BEGIN
	REGION read me
	  // ============================================================================
	  // PROGRAM START COMMENT
	  // ============================================================================
	  // EN:
	  // FC_AutoProcessPopup handles popup visualization and editing of AutoProcess
	  // data based on index from HMI.
	  // The function provides:
	  //  - automatic data loading from AutoProcessData according to selected index,
	  //  - two-step confirmation for safe data overwrite (compare first, write second),
	  //  - automatic reset of edit mode when index is changed,
	  //  - delete functionality for selected record,
	  //  - status bits for HMI to visualize pending changes and confirmation dialogs,
	  //  - index range control (1..16).
	  //
	  // Data flow:
	  // AutoProcessData  -> ActualSHowingData  (display mode)
	  // ActualSHowingData -> AutoProcessData  (after double confirmation)
	  //
	  // Usage:
	  // Call cyclically 
	  // RMS index is taken from AutoProcess_HMI.IndexProcess.
	  //
	  // ----------------------------------------------------------------------------
	  // CZ:
	  // FC_AutoProcessPopup obsluhuje zobrazení a editaci dat AutoProcess podle
	  // indexu z HMI.
	  // Funkce zajišťuje:
	  //  - automatické načítání dat z AutoProcessData podle zvoleného indexu,
	  //  - dvoukrokové potvrzení zápisu (nejprve porovnání, poté zápis),
	  //  - automatické zrušení editace při změně indexu,
	  //  - mazání záznamu podle indexu,
	  //  - stavové bity pro HMI (čekající změna, potvrzovací dialog),
	  //  - kontrolu rozsahu indexu (1..16).
	  //
	  // Tok dat:
	  // AutoProcessData  -> ActualSHowingData  (zobrazení)
	  // ActualSHowingData -> AutoProcessData  (po potvrzení)
	  //
	  // Použití:
	  // Volat cyklicky 
	  // Index je čten z AutoProcess_HMI.IndexProcess.
	  // ============================================================================
	  
	  // Statement section REGION
	  
	END_REGION
	
	
	REGION IndexRangeCheck
	  // EN: Clamp index to range 1..16
	  // CZ: Oříznutí indexu do rozsahu 1..16
	  IF #idx < 1 THEN
	    #idx := 1;
	    "AutoProcess_HMI".IndexProcess := #idx;
	  ELSIF #idx > 16 THEN
	    #idx := 16;
	    "AutoProcess_HMI".IndexProcess := #idx;
	    
	  END_IF;
	END_REGION
	
	
	REGION IndexHandling
	  // ---------------------------------------------------------------------------
	  // EN: Detect index change and reset edit session
	  // CZ: Detekce změny indexu a zrušení editace
	  // ---------------------------------------------------------------------------
	  #idx := "AutoProcess_HMI".IndexProcess;
	  
	  IF #idx <> "AutoProcess_HMI".Data_handling.LastIndex THEN
	    "AutoProcess_HMI".Data_handling.UpdateData_switch := FALSE;
	    "AutoProcess_HMI".Data_handling.UpdateData_Confirm := FALSE;
	    "AutoProcess_HMI".Data_handling.FinalConfirm_Write := FALSE;
	    "AutoProcess_HMI".Data_handling.ConfirmDialogActive := FALSE;
	    "AutoProcess_HMI".Data_handling.ChangePending := FALSE;
	    "AutoProcess_HMI".Data_handling.DeleteData := FALSE;
	    "AutoProcess_HMI".Data_handling.LastIndex := #idx;
	  END_IF;
	END_REGION
	
	
	
	REGION ShowData
	  // ---------------------------------------------------------------------------
	  // EN: Copy data to HMI if edit mode is inactive
	  // CZ: Zobrazování dat – pokud není editace, kopíruj data z DB
	  // ---------------------------------------------------------------------------
	  IF NOT "AutoProcess_HMI".Data_handling.UpdateData_switch THEN
	    CASE #idx OF
	      1:
	        "AutoProcess_HMI".ActualSHowingData := "AutoProcessData".A_ScanRotate;
	      2:
	        "AutoProcess_HMI".ActualSHowingData := "AutoProcessData".F_Robot1Grip1;
	      3:
	        "AutoProcess_HMI".ActualSHowingData := "AutoProcessData".F_Robot1Grip2;
	      4:
	        "AutoProcess_HMI".ActualSHowingData := "AutoProcessData".B_Press1;
	      5:
	        "AutoProcess_HMI".ActualSHowingData := "AutoProcessData".C_Glue;
	      6:
	        "AutoProcess_HMI".ActualSHowingData := "AutoProcessData".F_Robot2Grip1;
	      7:
	        "AutoProcess_HMI".ActualSHowingData := "AutoProcessData".F_Robot2Grip2;
	      8:
	        "AutoProcess_HMI".ActualSHowingData := "AutoProcessData".C_GlueNGBuffer;
	      9:
	        "AutoProcess_HMI".ActualSHowingData := "AutoProcessData".C_MagnScanNGBuffer;
	      10:
	        "AutoProcess_HMI".ActualSHowingData := "AutoProcessData".B_Press2;
	      11:
	        "AutoProcess_HMI".ActualSHowingData := "AutoProcessData".F_Robot3Grip1;
	      12:
	        "AutoProcess_HMI".ActualSHowingData := "AutoProcessData".F_Robot3Grip2;
	      13:
	        "AutoProcess_HMI".ActualSHowingData := "AutoProcessData".H_ShafeLine;
	      14:
	        "AutoProcess_HMI".ActualSHowingData := "AutoProcessData".J_ShafeLine;
	      15:
	        "AutoProcess_HMI".ActualSHowingData := "AutoProcessData".K_ShafeLine;
	      16:
	        "AutoProcess_HMI".ActualSHowingData := "AutoProcessData".L_ShafeLine;
	      ELSE
	        ;
	        // EN: invalid index / CZ: neplatný index
	    END_CASE;
	  END_IF;
	END_REGION
	
	
	
	REGION FirstConfirm
	  // ---------------------------------------------------------------------------
	  // EN: First confirmation → enable compare dialog
	  // CZ: První potvrzení → aktivace porovnávacího dialogu
	  // ---------------------------------------------------------------------------
	  IF "AutoProcess_HMI".Data_handling.UpdateData_switch
	    AND "AutoProcess_HMI".Data_handling.UpdateData_Confirm
	    AND NOT "AutoProcess_HMI".Data_handling.ConfirmDialogActive THEN
	    
	    "AutoProcess_HMI".Data_handling.ConfirmDialogActive := TRUE;
	    "AutoProcess_HMI".Data_handling.ChangePending := TRUE;
	    
	    "AutoProcess_HMI".Data_handling.UpdateData_Confirm := FALSE;
	  END_IF;
	END_REGION
	
	
	
	REGION FinalWrite
	  // ---------------------------------------------------------------------------
	  // EN: Final confirmation → write to data DB
	  // CZ: Finální potvrzení → zápis do DB
	  // ---------------------------------------------------------------------------
	  IF "AutoProcess_HMI".Data_handling.ConfirmDialogActive
	    AND "AutoProcess_HMI".Data_handling.FinalConfirm_Write THEN
	    
	    CASE #idx OF
	      1:
	        "AutoProcessData".A_ScanRotate := "AutoProcess_HMI".ActualSHowingData;
	      2:
	        "AutoProcessData".F_Robot1Grip1 := "AutoProcess_HMI".ActualSHowingData;
	      3:
	        "AutoProcessData".F_Robot1Grip2 := "AutoProcess_HMI".ActualSHowingData;
	      4:
	        "AutoProcessData".B_Press1 := "AutoProcess_HMI".ActualSHowingData;
	      5:
	        "AutoProcessData".C_Glue := "AutoProcess_HMI".ActualSHowingData;
	      6:
	        "AutoProcessData".F_Robot2Grip1 := "AutoProcess_HMI".ActualSHowingData;
	      7:
	        "AutoProcessData".F_Robot2Grip2 := "AutoProcess_HMI".ActualSHowingData;
	      8:
	        "AutoProcessData".C_GlueNGBuffer := "AutoProcess_HMI".ActualSHowingData;
	      9:
	        "AutoProcessData".C_MagnScanNGBuffer := "AutoProcess_HMI".ActualSHowingData;
	      10:
	        "AutoProcessData".B_Press2 := "AutoProcess_HMI".ActualSHowingData;
	      11:
	        "AutoProcessData".F_Robot3Grip1 := "AutoProcess_HMI".ActualSHowingData;
	      12:
	        "AutoProcessData".F_Robot3Grip2 := "AutoProcess_HMI".ActualSHowingData;
	      13:
	        "AutoProcessData".H_ShafeLine := "AutoProcess_HMI".ActualSHowingData;
	      14:
	        "AutoProcessData".J_ShafeLine := "AutoProcess_HMI".ActualSHowingData;
	      15:
	        "AutoProcessData".K_ShafeLine := "AutoProcess_HMI".ActualSHowingData;
	      16:
	        "AutoProcessData".L_ShafeLine := "AutoProcess_HMI".ActualSHowingData;
	      ELSE
	        ;
	    END_CASE;
	    
	    // reset flags after write
	    "AutoProcess_HMI".Data_handling.ConfirmDialogActive := FALSE;
	    "AutoProcess_HMI".Data_handling.ChangePending := FALSE;
	    "AutoProcess_HMI".Data_handling.FinalConfirm_Write := FALSE;
	    "AutoProcess_HMI".Data_handling.UpdateData_switch := FALSE;
	  END_IF;
	END_REGION
	
	
	
	REGION DeleteData
	  // ---------------------------------------------------------------------------
	  // EN: Delete selected Record (reset to default struct)
	  // CZ: Smazání záznamu – vynulování struktury
	  // ---------------------------------------------------------------------------
	  IF "AutoProcess_HMI".Data_handling.DeleteData AND
	    "AutoProcess_HMI".Data_handling.FinalConfirm_Write
	    THEN
	    
	    CASE #idx OF
	      1:
	        "AutoProcessData".A_ScanRotate := #DefaultData;
	      2:
	        "AutoProcessData".F_Robot1Grip1 := #DefaultData;
	      3:
	        "AutoProcessData".F_Robot1Grip2 := #DefaultData;
	      4:
	        "AutoProcessData".B_Press1 := #DefaultData;
	      5:
	        "AutoProcessData".C_Glue := #DefaultData;
	      6:
	        "AutoProcessData".F_Robot2Grip1 := #DefaultData;
	      7:
	        "AutoProcessData".F_Robot2Grip2 := #DefaultData;
	      8:
	        "AutoProcessData".C_GlueNGBuffer := #DefaultData;
	      9:
	        "AutoProcessData".C_MagnScanNGBuffer := #DefaultData;
	      10:
	        "AutoProcessData".B_Press2 := #DefaultData;
	      11:
	        "AutoProcessData".F_Robot3Grip1 := #DefaultData;
	      12:
	        "AutoProcessData".F_Robot3Grip2 := #DefaultData;
	      13:
	        "AutoProcessData".H_ShafeLine := #DefaultData;
	      14:
	        "AutoProcessData".J_ShafeLine := #DefaultData;
	      15:
	        "AutoProcessData".K_ShafeLine := #DefaultData;
	      16:
	        "AutoProcessData".L_ShafeLine := #DefaultData;
	      ELSE
	        ;
	    END_CASE;
	    
	    // reset delete + editing states
	    "AutoProcess_HMI".Data_handling.DeleteData := FALSE;
	    "AutoProcess_HMI".Data_handling.UpdateData_switch := FALSE;
	    "AutoProcess_HMI".Data_handling.UpdateData_Confirm := FALSE;
	    "AutoProcess_HMI".Data_handling.FinalConfirm_Write := FALSE;
	    "AutoProcess_HMI".Data_handling.ConfirmDialogActive := FALSE;
	    "AutoProcess_HMI".Data_handling.ChangePending := FALSE;
	  END_IF;
	END_REGION
	
	REGION StationProductIcons
	  // EN: Set icon bits if station contains product (PartStatus <> 0)
	  // CZ: Nastavení bitů ikony – stanice má kus, pokud PartStatus <> 0
	  
	  // 1 – A_ScanRotate
	  "AutoProcess_HMI".StationHasProduct[1] :=
	  "AutoProcessData".A_ScanRotate.PartStatus <> 0;
	  
	  // 2 – F_Robot1Grip1
	  "AutoProcess_HMI".StationHasProduct[2] :=
	  "AutoProcessData".F_Robot1Grip1.PartStatus <> 0;
	  
	  // 3 – F_Robot1Grip2
	  "AutoProcess_HMI".StationHasProduct[3] :=
	  "AutoProcessData".F_Robot1Grip2.PartStatus <> 0;
	  
	  // 4 – B_Press1
	  "AutoProcess_HMI".StationHasProduct[4] :=
	  "AutoProcessData".B_Press1.PartStatus <> 0;
	  
	  // 5 – C_Glue
	  "AutoProcess_HMI".StationHasProduct[5] :=
	  "AutoProcessData".C_Glue.PartStatus <> 0;
	  
	  // 6 – F_Robot2Grip1
	  "AutoProcess_HMI".StationHasProduct[6] :=
	  "AutoProcessData".F_Robot2Grip1.PartStatus <> 0;
	  
	  // 7 – F_Robot2Grip2
	  "AutoProcess_HMI".StationHasProduct[7] :=
	  "AutoProcessData".F_Robot2Grip2.PartStatus <> 0;
	  
	  // 8 – C_GlueNGBuffer
	  "AutoProcess_HMI".StationHasProduct[8] :=
	  "AutoProcessData".C_GlueNGBuffer.PartStatus <> 0;
	  
	  // 9 – C_MagnScanNGBuffer
	  "AutoProcess_HMI".StationHasProduct[9] :=
	  "AutoProcessData".C_MagnScanNGBuffer.PartStatus <> 0;
	  
	  // 10 – B_Press2
	  "AutoProcess_HMI".StationHasProduct[10] :=
	  "AutoProcessData".B_Press2.PartStatus <> 0;
	  
	  // 11 – F_Robot3Grip1
	  "AutoProcess_HMI".StationHasProduct[11] :=
	  "AutoProcessData".F_Robot3Grip1.PartStatus <> 0;
	  
	  // 12 – F_Robot3Grip2
	  "AutoProcess_HMI".StationHasProduct[12] :=
	  "AutoProcessData".F_Robot3Grip2.PartStatus <> 0;
	  
	  // 13 – H_ShafeLine
	  "AutoProcess_HMI".StationHasProduct[13] :=
	  "AutoProcessData".H_ShafeLine.PartStatus <> 0;
	  
	  // 14 – J_ShafeLine
	  "AutoProcess_HMI".StationHasProduct[14] :=
	  "AutoProcessData".J_ShafeLine.PartStatus <> 0;
	  
	  // 15 – K_ShafeLine
	  "AutoProcess_HMI".StationHasProduct[15] :=
	  "AutoProcessData".K_ShafeLine.PartStatus <> 0;
	  
	  // 16 – L_ShafeLine
	  "AutoProcess_HMI".StationHasProduct[16] :=
	  "AutoProcessData".L_ShafeLine.PartStatus <> 0;
	  
	END_REGION
	
	
END_FUNCTION_BLOCK

ORGANIZATION_BLOCK "03_CYC_INT2"   // OB32, LAD, CyclicInterrupt
TITLE = "Cyclic Interrupt"
{ S7_Optimized_Access := 'FALSE' }
// stored: AutoNumber false, SetENOAutomatically false
   VAR_TEMP
      OB32_EV_CLASS : Byte;   // Bits 0-3 = 1 (Coming event), Bits 4-7 = 1 (Event class 1)
      OB32_STRT_INF : Byte;   // 16#33 (OB 32 has started)
      OB32_PRIORITY : Byte;   // Priority of OB Execution
      OB32_OB_NUMBR : Byte;   // 32 (Organization block 32, OB32)
      OB32_RESERVED_1 : Byte;   // Reserved for system
      OB32_RESERVED_2 : Byte;   // Reserved for system
      OB32_PHS_OFFSET : Int;   // Phase offset (integer, milliseconds)
      OB32_RESERVED_3 : Int;   // Reserved for system
      OB32_EXC_FREQ : Int;   // Frequency of execution (msec)
      OB32_DATE_TIME : Date_And_Time;   // Date and time OB32 started
   END_VAR
BEGIN

REGION Network 1
   // //Keep resource code
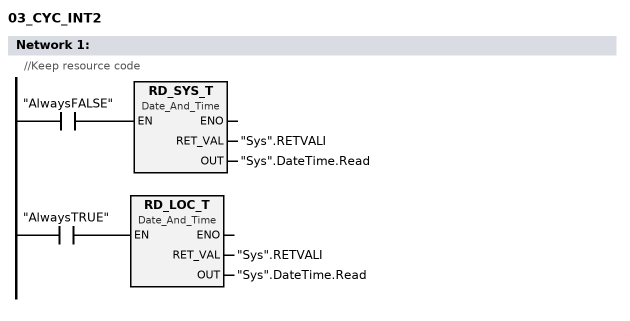
   RUNG wire#powerrail
      Contact( "AlwaysFALSE" )
      { S7_Templates := "date_type := Date_And_Time" } RD_SYS_T(RET_VAL => "Sys".RETVALI, OUT => "Sys".DateTime.Read)
   END_RUNG
   RUNG wire#powerrail
      Contact( "AlwaysTRUE" )
      { S7_Templates := "date_type := Date_And_Time" } RD_LOC_T(RET_VAL => "Sys".RETVALI, OUT => "Sys".DateTime.Read)
   END_RUNG
   // the same network as SCL:
   IF "AlwaysFALSE" THEN "Sys".RETVALI := RD_SYS_T(OUT => "Sys".DateTime.Read); END_IF;
   IF "AlwaysTRUE" THEN "Sys".RETVALI := RD_LOC_T(OUT => "Sys".DateTime.Read); END_IF;
END_REGION

NETWORK
TITLE = Diagnostic
//      CALL  "Diagnostic"
//         iCPUType :=2
//         iDBNum   :=3001
//         iOffset  :=0


END_ORGANIZATION_BLOCK

ORGANIZATION_BLOCK "04_CYC_INT5"   // OB35, LAD, CyclicInterrupt
TITLE = "Cyclic Interrupt"
{ S7_Optimized_Access := 'FALSE' }
// stored: AutoNumber false, SetENOAutomatically false
   VAR_TEMP
      OB35_EV_CLASS : Byte;   // Bits 0-3 = 1 (Coming event), Bits 4-7 = 1 (Event class 1)
      OB35_STRT_INF : Byte;   // 16#36 (OB 35 has started)
      OB35_PRIORITY : Byte;   // Priority of OB Execution
      OB35_OB_NUMBR : Byte;   // 35 (Organization block 35, OB35)
      OB35_RESERVED_1 : Byte;   // Reserved for system
      OB35_RESERVED_2 : Byte;   // Reserved for system
      OB35_PHASE_OFFSET : Word;   // Phase offset (msec)
      OB35_RESERVED_3 : Int;   // Reserved for system
      OB35_EXC_FREQ : Int;   // Frequency of execution (msec)
      OB35_DATE_TIME : Date_And_Time;   // Date and time OB35 started
   END_VAR
BEGIN
END_ORGANIZATION_BLOCK

FUNCTION_BLOCK "MaterialGate"   // FB5210, LAD
{ S7_Optimized_Access := 'FALSE' }
// stored: AutoNumber false, SetENOAutomatically false
   VAR_INPUT
      iSysInface : "RCS_SysComInterface_V1";
      "iMaterialGate Opened Monitor" : Bool;   // 安全门打开状态监控
      "iMaterialGate Locked Monitor" : Bool;   // 安全门锁定状态监控
      i1s_Pulse : Bool;   // 1s脉冲信号
      "iMaterialGate AutoLock Timer" : Time := T#1s;   // 安全门自动模式下锁延时
      "iMaterialGate ManualLock Timer" : Time := T#60s;   // 安全门手动模式下锁定延时
   END_VAR
   VAR_OUTPUT
      "oMaterialGate LockedLamp" { ExternalAccessible := 'False'; ExternalVisible := 'False'; ExternalWritable := 'False'} : Bool;   // 安全门解锁输出状态
   END_VAR
   VAR_IN_OUT
      ioMaterialGateLock : Bool;   // 安全门锁定输出
      ioHMI_Interface : "SafetyGateUDT";
   END_VAR
   VAR
      "sMaterialafetyGate Timer" { S7_SetPoint := 'True'} : Array[1..5] of TON_TIME;
      sP_Trig : Array[1..10] of Bool;
      sN_Trig : Array[1..10] of Bool;
      "sMaterialGate UnlockRequest" { ExternalAccessible := 'False'; ExternalVisible := 'False'; ExternalWritable := 'False'} : Bool;   // 安全门开门请求标志位
      "sMaterialGate LockRequest" : Bool;
   END_VAR
   VAR_TEMP
      tAlyways_On : Bool;
      tAlyways_Off : Bool;
   END_VAR
   VAR_TEMP   // added for the SCL form of the ladder/FBD networks
      _w1 : Bool;
      _w2 : Bool;
      _w3 : Bool;
      _w4 : Bool;
      _w5 : Bool;
      _w6 : Bool;
      _w7 : Bool;
   END_VAR
BEGIN

REGION Network 1: #tAlyways_On
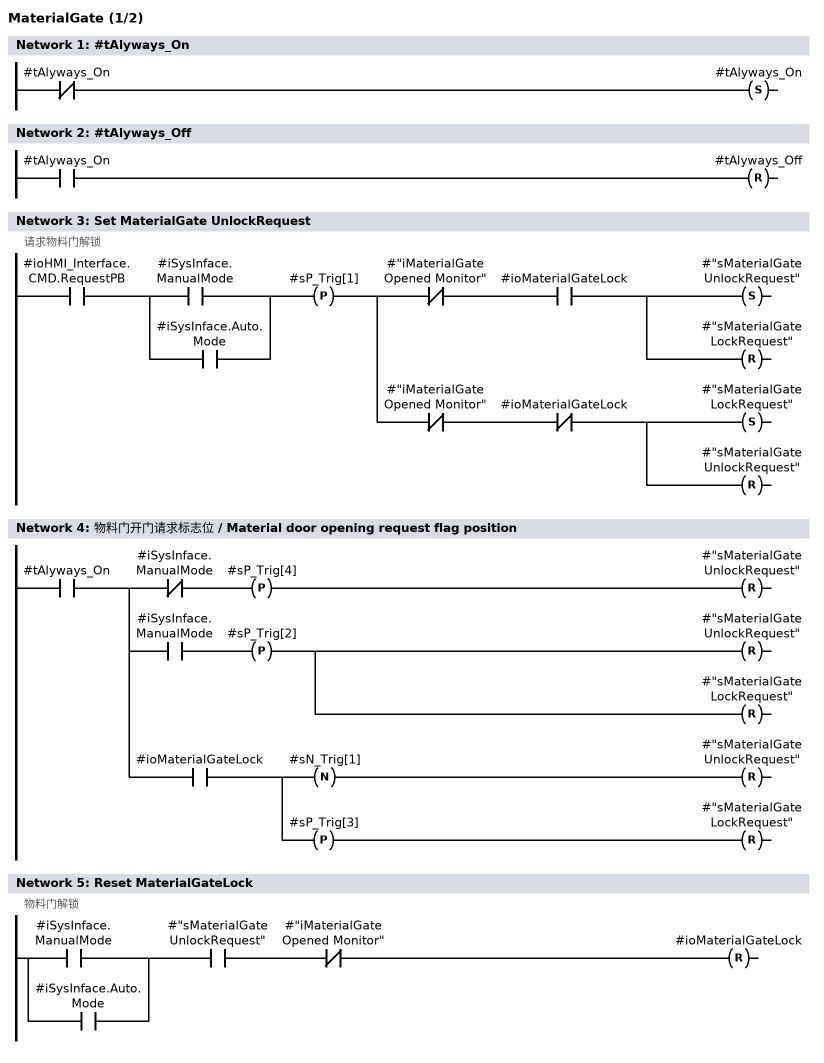
   RUNG wire#powerrail
      I_Contact( #tAlyways_On )
      S_Coil( #tAlyways_On )
   END_RUNG
   // the same network as SCL:
   IF NOT #tAlyways_On THEN #tAlyways_On := TRUE; END_IF;
END_REGION

REGION Network 2: #tAlyways_Off
   RUNG wire#powerrail
      Contact( #tAlyways_On )
      R_Coil( #tAlyways_Off )
   END_RUNG
   // the same network as SCL:
   IF #tAlyways_On THEN #tAlyways_Off := FALSE; END_IF;
END_REGION

REGION Network 3: Set MaterialGate UnlockRequest
   // 请求物料门解锁
   RUNG wire#powerrail
      Contact( #ioHMI_Interface.CMD.RequestPB )
      wire#w1
      Contact( #iSysInface.ManualMode )
      wire#w2
      P_Trig( #sP_Trig[1] )
      wire#w3
      I_Contact( #"iMaterialGate Opened Monitor" )
      Contact( #ioMaterialGateLock )
      wire#w4
      S_Coil( #"sMaterialGate UnlockRequest" )
   END_RUNG
   RUNG wire#w1
      Contact( #iSysInface.Auto.Mode )
   END_RUNG wire#w2
   RUNG wire#w4
      R_Coil( #"sMaterialGate LockRequest" )
   END_RUNG
   RUNG wire#w3
      I_Contact( #"iMaterialGate Opened Monitor" )
      I_Contact( #ioMaterialGateLock )
      wire#w5
      S_Coil( #"sMaterialGate LockRequest" )
   END_RUNG
   RUNG wire#w5
      R_Coil( #"sMaterialGate UnlockRequest" )
   END_RUNG
   // the same network as SCL:
   #_w1 := #ioHMI_Interface.CMD.RequestPB AND (#iSysInface.ManualMode OR #iSysInface.Auto.Mode);
   #_w2 := #_w1 AND NOT #sP_Trig[1];   // rising edge
   #sP_Trig[1] := #_w1;
   IF #_w2 AND NOT #"iMaterialGate Opened Monitor" AND #ioMaterialGateLock THEN
       #"sMaterialGate UnlockRequest" := TRUE;
       #"sMaterialGate LockRequest" := FALSE;
   END_IF;
   IF #_w2 AND NOT #"iMaterialGate Opened Monitor" AND NOT #ioMaterialGateLock THEN
       #"sMaterialGate LockRequest" := TRUE;
       #"sMaterialGate UnlockRequest" := FALSE;
   END_IF;
END_REGION

REGION Network 4: 物料门开门请求标志位 / Material door opening request flag position
   RUNG wire#powerrail
      Contact( #tAlyways_On )
      wire#w1
      I_Contact( #iSysInface.ManualMode )
      P_Trig( #sP_Trig[4] )
      R_Coil( #"sMaterialGate UnlockRequest" )
   END_RUNG
   RUNG wire#w1
      Contact( #iSysInface.ManualMode )
      P_Trig( #sP_Trig[2] )
      wire#w2
      R_Coil( #"sMaterialGate UnlockRequest" )
   END_RUNG
   RUNG wire#w2
      R_Coil( #"sMaterialGate LockRequest" )
   END_RUNG
   RUNG wire#w1
      Contact( #ioMaterialGateLock )
      wire#w3
      N_Trig( #sN_Trig[1] )
      R_Coil( #"sMaterialGate UnlockRequest" )
   END_RUNG
   RUNG wire#w3
      P_Trig( #sP_Trig[3] )
      R_Coil( #"sMaterialGate LockRequest" )
   END_RUNG
   // the same network as SCL:
   #_w1 := #tAlyways_On AND NOT #iSysInface.ManualMode;
   #_w2 := #_w1 AND NOT #sP_Trig[4];   // rising edge
   #sP_Trig[4] := #_w1;
   IF #_w2 THEN #"sMaterialGate UnlockRequest" := FALSE; END_IF;
   #_w3 := #tAlyways_On AND #iSysInface.ManualMode;
   #_w4 := #_w3 AND NOT #sP_Trig[2];   // rising edge
   #sP_Trig[2] := #_w3;
   IF #_w4 THEN
       #"sMaterialGate UnlockRequest" := FALSE;
       #"sMaterialGate LockRequest" := FALSE;
   END_IF;
   #_w5 := #tAlyways_On AND #ioMaterialGateLock;
   #_w6 := NOT #_w5 AND #sN_Trig[1];   // falling edge
   #sN_Trig[1] := #_w5;
   IF #_w6 THEN #"sMaterialGate UnlockRequest" := FALSE; END_IF;
   #_w7 := #_w5 AND NOT #sP_Trig[3];   // rising edge
   #sP_Trig[3] := #_w5;
   IF #_w7 THEN #"sMaterialGate LockRequest" := FALSE; END_IF;
END_REGION

REGION Network 5: Reset MaterialGateLock
   // 物料门解锁
   RUNG wire#powerrail
      Contact( #iSysInface.ManualMode )
      wire#w1
      Contact( #"sMaterialGate UnlockRequest" )
      I_Contact( #"iMaterialGate Opened Monitor" )
      R_Coil( #ioMaterialGateLock )
   END_RUNG
   RUNG wire#powerrail
      Contact( #iSysInface.Auto.Mode )
   END_RUNG wire#w1
   // the same network as SCL:
   IF (#iSysInface.ManualMode OR #iSysInface.Auto.Mode) AND #"sMaterialGate UnlockRequest" AND NOT #"iMaterialGate Opened Monitor" THEN
       #ioMaterialGateLock := FALSE;
   END_IF;
END_REGION

REGION Network 6: Set MaterialGate Lock
   // 物料门锁定
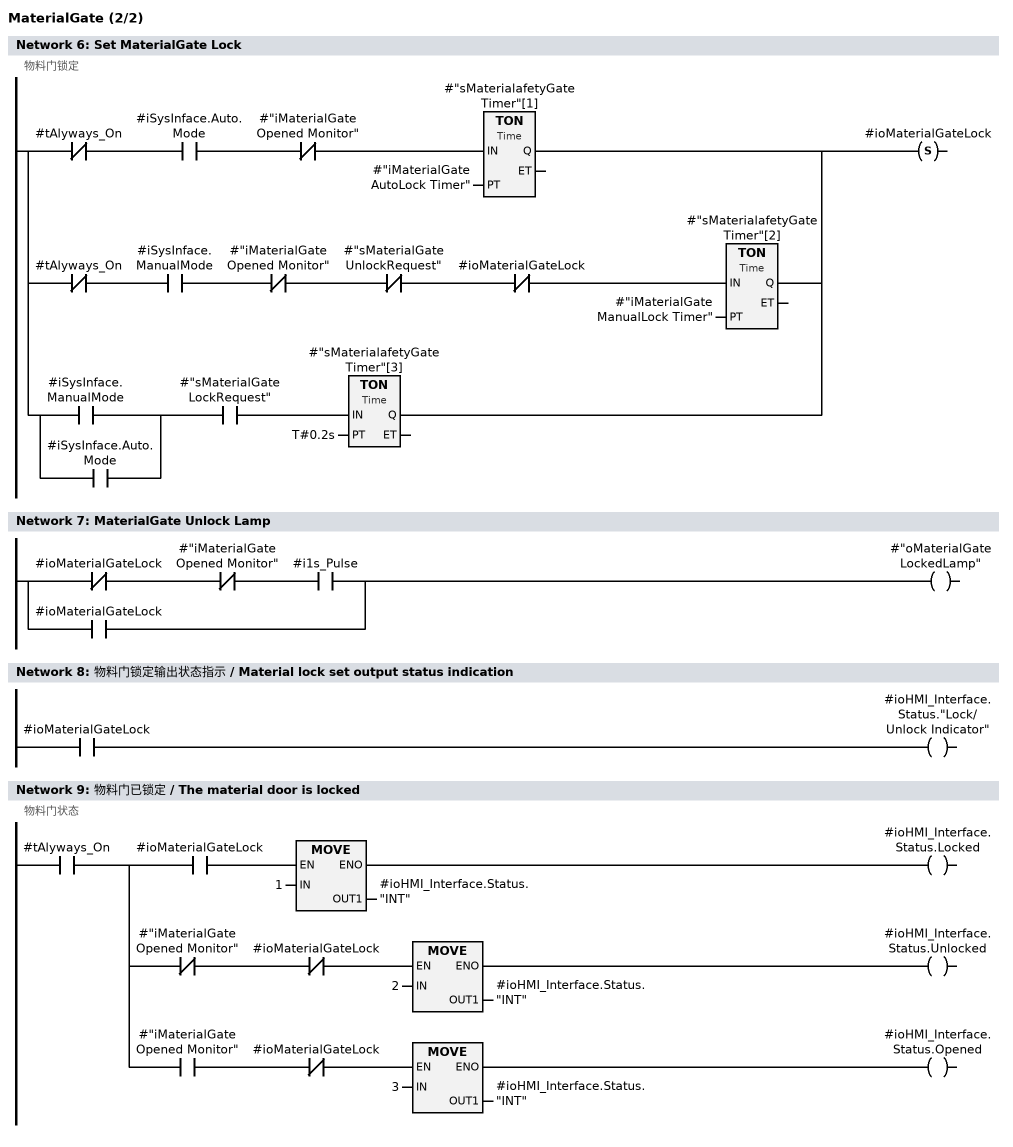
   RUNG wire#powerrail
      I_Contact( #tAlyways_On )
      Contact( #iSysInface.Auto.Mode )
      I_Contact( #"iMaterialGate Opened Monitor" )
      { S7_Templates := "time_type := Time" } #"sMaterialafetyGate Timer"[1].TON(pt := #"iMaterialGate AutoLock Timer", et =>)
      wire#w1
      S_Coil( #ioMaterialGateLock )
   END_RUNG
   RUNG wire#powerrail
      I_Contact( #tAlyways_On )
      Contact( #iSysInface.ManualMode )
      I_Contact( #"iMaterialGate Opened Monitor" )
      I_Contact( #"sMaterialGate UnlockRequest" )
      I_Contact( #ioMaterialGateLock )
      { S7_Templates := "time_type := Time" } #"sMaterialafetyGate Timer"[2].TON(pt := #"iMaterialGate ManualLock Timer", et =>)
   END_RUNG wire#w1
   RUNG wire#powerrail
      Contact( #iSysInface.ManualMode )
      wire#w2
      Contact( #"sMaterialGate LockRequest" )
      { S7_Templates := "time_type := Time" } #"sMaterialafetyGate Timer"[3].TON(pt := T#0.2s, et =>)
   END_RUNG wire#w1
   RUNG wire#powerrail
      Contact( #iSysInface.Auto.Mode )
   END_RUNG wire#w2
   // the same network as SCL:
   #"sMaterialafetyGate Timer"[1].TON(IN := NOT #tAlyways_On AND #iSysInface.Auto.Mode AND NOT #"iMaterialGate Opened Monitor",
                           PT := #"iMaterialGate AutoLock Timer");
   #_w1 := #"sMaterialafetyGate Timer"[1].Q;
   #"sMaterialafetyGate Timer"[2].TON(IN := NOT #tAlyways_On AND #iSysInface.ManualMode AND NOT #"iMaterialGate Opened Monitor" AND NOT #"sMaterialGate UnlockRequest" AND NOT #ioMaterialGateLock,
                           PT := #"iMaterialGate ManualLock Timer");
   #_w2 := #"sMaterialafetyGate Timer"[2].Q;
   #"sMaterialafetyGate Timer"[3].TON(IN := (#iSysInface.ManualMode OR #iSysInface.Auto.Mode) AND #"sMaterialGate LockRequest",
                           PT := T#0.2s);
   IF #_w1 OR #_w2 OR #"sMaterialafetyGate Timer"[3].Q THEN #ioMaterialGateLock := TRUE; END_IF;
END_REGION

REGION Network 7: MaterialGate Unlock Lamp
   RUNG wire#powerrail
      I_Contact( #ioMaterialGateLock )
      I_Contact( #"iMaterialGate Opened Monitor" )
      Contact( #i1s_Pulse )
      wire#w1
      Coil( #"oMaterialGate LockedLamp" )
   END_RUNG
   RUNG wire#powerrail
      Contact( #ioMaterialGateLock )
   END_RUNG wire#w1
   // the same network as SCL:
   #"oMaterialGate LockedLamp" := (NOT #ioMaterialGateLock AND NOT #"iMaterialGate Opened Monitor" AND #i1s_Pulse) OR #ioMaterialGateLock;
END_REGION

REGION Network 8: 物料门锁定输出状态指示 / Material lock set output status indication
   RUNG wire#powerrail
      Contact( #ioMaterialGateLock )
      Coil( #ioHMI_Interface.Status."Lock/Unlock Indicator" )
   END_RUNG
   // the same network as SCL:
   #ioHMI_Interface.Status."Lock/Unlock Indicator" := #ioMaterialGateLock;
END_REGION

REGION Network 9: 物料门已锁定 / The material door is locked
   // 物料门状态
   RUNG wire#powerrail
      Contact( #tAlyways_On )
      wire#w1
      Contact( #ioMaterialGateLock )
      Move(in := 1, out1 => #ioHMI_Interface.Status."INT")
      Coil( #ioHMI_Interface.Status.Locked )
   END_RUNG
   RUNG wire#w1
      I_Contact( #"iMaterialGate Opened Monitor" )
      I_Contact( #ioMaterialGateLock )
      Move(in := 2, out1 => #ioHMI_Interface.Status."INT")
      Coil( #ioHMI_Interface.Status.Unlocked )
   END_RUNG
   RUNG wire#w1
      Contact( #"iMaterialGate Opened Monitor" )
      I_Contact( #ioMaterialGateLock )
      Move(in := 3, out1 => #ioHMI_Interface.Status."INT")
      Coil( #ioHMI_Interface.Status.Opened )
   END_RUNG
   // the same network as SCL:
   #_w1 := #tAlyways_On AND #ioMaterialGateLock;
   IF #_w1 THEN #ioHMI_Interface.Status."INT" := 1; END_IF;
   #ioHMI_Interface.Status.Locked := #_w1;
   #_w2 := #tAlyways_On AND NOT #"iMaterialGate Opened Monitor" AND NOT #ioMaterialGateLock;
   IF #_w2 THEN #ioHMI_Interface.Status."INT" := 2; END_IF;
   #ioHMI_Interface.Status.Unlocked := #_w2;
   #_w3 := #tAlyways_On AND #"iMaterialGate Opened Monitor" AND NOT #ioMaterialGateLock;
   IF #_w3 THEN #ioHMI_Interface.Status."INT" := 3; END_IF;
   #ioHMI_Interface.Status.Opened := #_w3;
END_REGION
END_FUNCTION_BLOCK

FUNCTION "ChangeOverProcess" : Void   // FC1000, LAD
{ S7_Optimized_Access := 'TRUE' }
// stored: AutoNumber false, SetENOAutomatically false
   VAR_TEMP
      tBool : Bool;
   END_VAR
   VAR_TEMP   // added for the SCL form of the ladder/FBD networks
      _w1 : Bool;
      _w2 : Bool;
      _w3 : Bool;
      _w4 : Bool;
      _w5 : Bool;
      _w6 : Bool;
      _w7 : Bool;
      _w8 : Bool;
   END_VAR
BEGIN

REGION Network 1: HMI ChangeOver Confirm
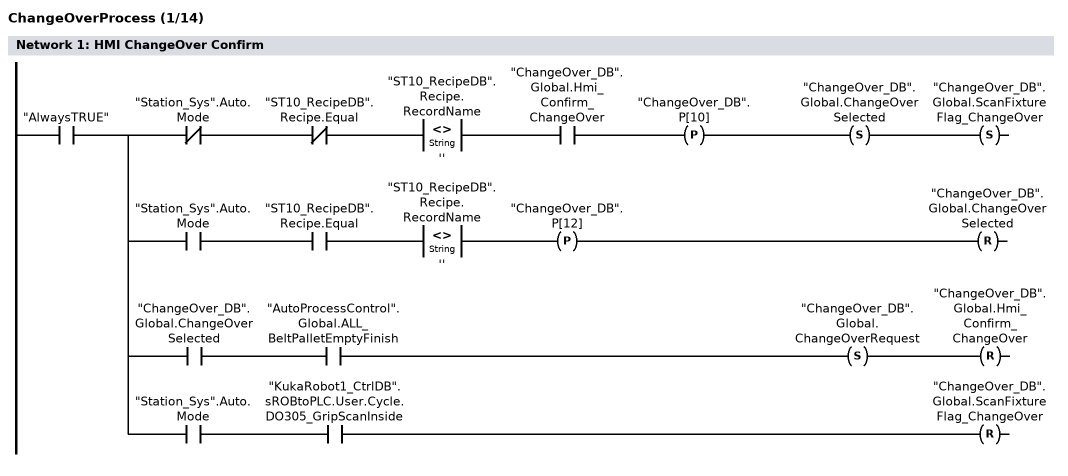
   RUNG wire#powerrail
      Contact( "AlwaysTRUE" )
      wire#w1
      I_Contact( "Station_Sys".Auto.Mode )
      I_Contact( "ST10_RecipeDB".Recipe.Equal )
      { S7_Templates := "SrcType := String" } NE_Contact(in1 := "ST10_RecipeDB".Recipe.RecordName, in2 := '')
      Contact( "ChangeOver_DB".Global.Hmi_Confirm_ChangeOver )
      P_Trig( "ChangeOver_DB".P[10] )
      S_Coil( "ChangeOver_DB".Global.ChangeOverSelected )
      S_Coil( "ChangeOver_DB".Global.ScanFixtureFlag_ChangeOver )
   END_RUNG
   RUNG wire#w1
      Contact( "Station_Sys".Auto.Mode )
      Contact( "ST10_RecipeDB".Recipe.Equal )
      { S7_Templates := "SrcType := String" } NE_Contact(in1 := "ST10_RecipeDB".Recipe.RecordName, in2 := '')
      P_Trig( "ChangeOver_DB".P[12] )
      R_Coil( "ChangeOver_DB".Global.ChangeOverSelected )
   END_RUNG
   RUNG wire#w1
      Contact( "ChangeOver_DB".Global.ChangeOverSelected )
      Contact( "AutoProcessControl".Global.ALL_BeltPalletEmptyFinish )
      S_Coil( "ChangeOver_DB".Global.ChangeOverRequest )
      R_Coil( "ChangeOver_DB".Global.Hmi_Confirm_ChangeOver )
   END_RUNG
   RUNG wire#w1
      Contact( "Station_Sys".Auto.Mode )
      Contact( "KukaRobot1_CtrlDB".sROBtoPLC.User.Cycle.DO305_GripScanInside )
      R_Coil( "ChangeOver_DB".Global.ScanFixtureFlag_ChangeOver )
   END_RUNG
   // the same network as SCL:
   #_w1 := "AlwaysTRUE" AND NOT "Station_Sys".Auto.Mode AND NOT "ST10_RecipeDB".Recipe.Equal AND ("ST10_RecipeDB".Recipe.RecordName <> '') AND "ChangeOver_DB".Global.Hmi_Confirm_ChangeOver;
   #_w2 := #_w1 AND NOT "ChangeOver_DB".P[10];   // rising edge
   "ChangeOver_DB".P[10] := #_w1;
   IF #_w2 THEN
       "ChangeOver_DB".Global.ChangeOverSelected := TRUE;
       "ChangeOver_DB".Global.ScanFixtureFlag_ChangeOver := TRUE;
   END_IF;
   #_w3 := "AlwaysTRUE" AND "Station_Sys".Auto.Mode AND "ST10_RecipeDB".Recipe.Equal AND ("ST10_RecipeDB".Recipe.RecordName <> '');
   #_w4 := #_w3 AND NOT "ChangeOver_DB".P[12];   // rising edge
   "ChangeOver_DB".P[12] := #_w3;
   IF #_w4 THEN "ChangeOver_DB".Global.ChangeOverSelected := FALSE; END_IF;
   IF "AlwaysTRUE" AND "ChangeOver_DB".Global.ChangeOverSelected AND "AutoProcessControl".Global.ALL_BeltPalletEmptyFinish THEN
       "ChangeOver_DB".Global.ChangeOverRequest := TRUE;
       "ChangeOver_DB".Global.Hmi_Confirm_ChangeOver := FALSE;
   END_IF;
   IF "AlwaysTRUE" AND "Station_Sys".Auto.Mode AND "KukaRobot1_CtrlDB".sROBtoPLC.User.Cycle.DO305_GripScanInside THEN
       "ChangeOver_DB".Global.ScanFixtureFlag_ChangeOver := FALSE;
   END_IF;
END_REGION

REGION Network 2: ChangeOverFinish Reset
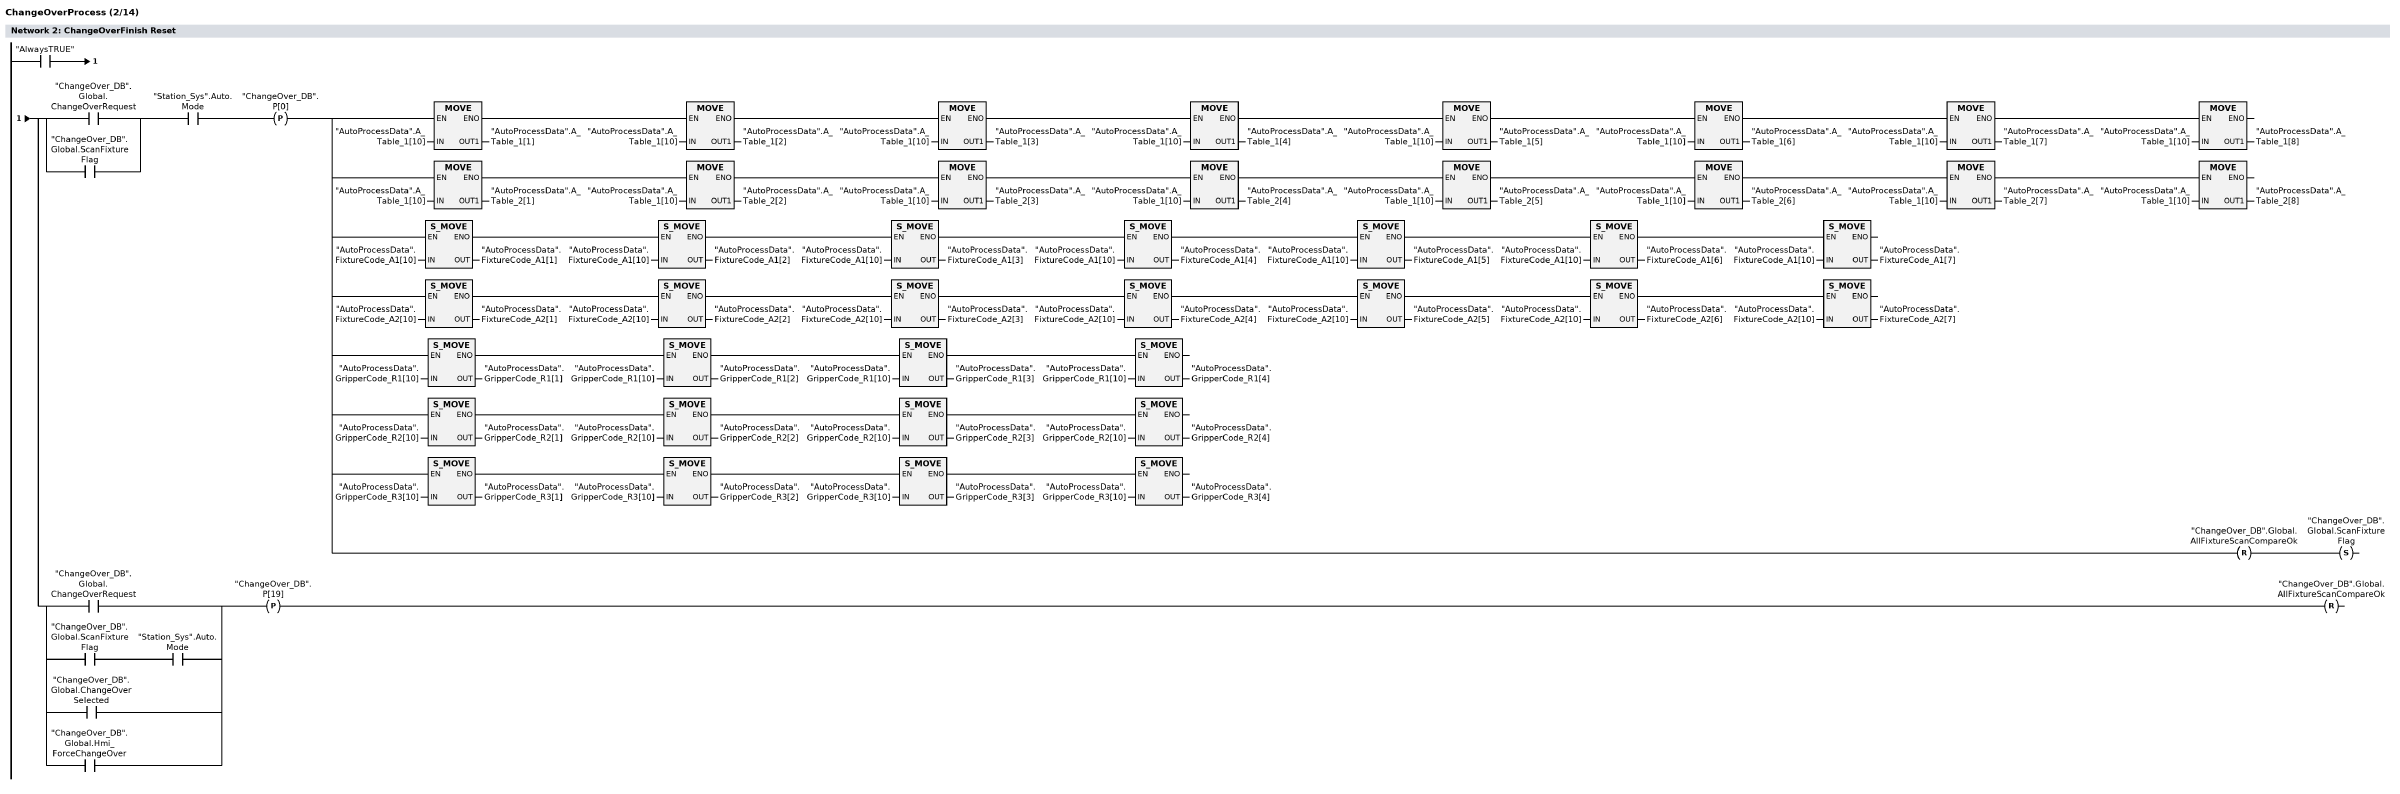
   RUNG wire#powerrail
      Contact( "AlwaysTRUE" )
      wire#w1
      Contact( "ChangeOver_DB".Global.ChangeOverRequest )
      wire#w2
      Contact( "Station_Sys".Auto.Mode )
      P_Trig( "ChangeOver_DB".P[0] )
      wire#w3
      Move(in := "AutoProcessData".A_Table_1[10], out1 => "AutoProcessData".A_Table_1[1])
      Move(in := "AutoProcessData".A_Table_1[10], out1 => "AutoProcessData".A_Table_1[2])
      Move(in := "AutoProcessData".A_Table_1[10], out1 => "AutoProcessData".A_Table_1[3])
      Move(in := "AutoProcessData".A_Table_1[10], out1 => "AutoProcessData".A_Table_1[4])
      Move(in := "AutoProcessData".A_Table_1[10], out1 => "AutoProcessData".A_Table_1[5])
      Move(in := "AutoProcessData".A_Table_1[10], out1 => "AutoProcessData".A_Table_1[6])
      Move(in := "AutoProcessData".A_Table_1[10], out1 => "AutoProcessData".A_Table_1[7])
      Move(in := "AutoProcessData".A_Table_1[10], out1 => "AutoProcessData".A_Table_1[8])
   END_RUNG
   RUNG wire#w1
      Contact( "ChangeOver_DB".Global.ScanFixtureFlag )
   END_RUNG wire#w2
   RUNG wire#w3
      Move(in := "AutoProcessData".A_Table_1[10], out1 => "AutoProcessData".A_Table_2[1])
      Move(in := "AutoProcessData".A_Table_1[10], out1 => "AutoProcessData".A_Table_2[2])
      Move(in := "AutoProcessData".A_Table_1[10], out1 => "AutoProcessData".A_Table_2[3])
      Move(in := "AutoProcessData".A_Table_1[10], out1 => "AutoProcessData".A_Table_2[4])
      Move(in := "AutoProcessData".A_Table_1[10], out1 => "AutoProcessData".A_Table_2[5])
      Move(in := "AutoProcessData".A_Table_1[10], out1 => "AutoProcessData".A_Table_2[6])
      Move(in := "AutoProcessData".A_Table_1[10], out1 => "AutoProcessData".A_Table_2[7])
      Move(in := "AutoProcessData".A_Table_1[10], out1 => "AutoProcessData".A_Table_2[8])
   END_RUNG
   RUNG wire#w3
      S_Move(in := "AutoProcessData".FixtureCode_A1[10], out => "AutoProcessData".FixtureCode_A1[1])
      S_Move(in := "AutoProcessData".FixtureCode_A1[10], out => "AutoProcessData".FixtureCode_A1[2])
      S_Move(in := "AutoProcessData".FixtureCode_A1[10], out => "AutoProcessData".FixtureCode_A1[3])
      S_Move(in := "AutoProcessData".FixtureCode_A1[10], out => "AutoProcessData".FixtureCode_A1[4])
      S_Move(in := "AutoProcessData".FixtureCode_A1[10], out => "AutoProcessData".FixtureCode_A1[5])
      S_Move(in := "AutoProcessData".FixtureCode_A1[10], out => "AutoProcessData".FixtureCode_A1[6])
      S_Move(in := "AutoProcessData".FixtureCode_A1[10], out => "AutoProcessData".FixtureCode_A1[7])
   END_RUNG
   RUNG wire#w3
      S_Move(in := "AutoProcessData".FixtureCode_A2[10], out => "AutoProcessData".FixtureCode_A2[1])
      S_Move(in := "AutoProcessData".FixtureCode_A2[10], out => "AutoProcessData".FixtureCode_A2[2])
      S_Move(in := "AutoProcessData".FixtureCode_A2[10], out => "AutoProcessData".FixtureCode_A2[3])
      S_Move(in := "AutoProcessData".FixtureCode_A2[10], out => "AutoProcessData".FixtureCode_A2[4])
      S_Move(in := "AutoProcessData".FixtureCode_A2[10], out => "AutoProcessData".FixtureCode_A2[5])
      S_Move(in := "AutoProcessData".FixtureCode_A2[10], out => "AutoProcessData".FixtureCode_A2[6])
      S_Move(in := "AutoProcessData".FixtureCode_A2[10], out => "AutoProcessData".FixtureCode_A2[7])
   END_RUNG
   RUNG wire#w3
      S_Move(in := "AutoProcessData".GripperCode_R1[10], out => "AutoProcessData".GripperCode_R1[1])
      S_Move(in := "AutoProcessData".GripperCode_R1[10], out => "AutoProcessData".GripperCode_R1[2])
      S_Move(in := "AutoProcessData".GripperCode_R1[10], out => "AutoProcessData".GripperCode_R1[3])
      S_Move(in := "AutoProcessData".GripperCode_R1[10], out => "AutoProcessData".GripperCode_R1[4])
   END_RUNG
   RUNG wire#w3
      S_Move(in := "AutoProcessData".GripperCode_R2[10], out => "AutoProcessData".GripperCode_R2[1])
      S_Move(in := "AutoProcessData".GripperCode_R2[10], out => "AutoProcessData".GripperCode_R2[2])
      S_Move(in := "AutoProcessData".GripperCode_R2[10], out => "AutoProcessData".GripperCode_R2[3])
      S_Move(in := "AutoProcessData".GripperCode_R2[10], out => "AutoProcessData".GripperCode_R2[4])
   END_RUNG
   RUNG wire#w3
      S_Move(in := "AutoProcessData".GripperCode_R3[10], out => "AutoProcessData".GripperCode_R3[1])
      S_Move(in := "AutoProcessData".GripperCode_R3[10], out => "AutoProcessData".GripperCode_R3[2])
      S_Move(in := "AutoProcessData".GripperCode_R3[10], out => "AutoProcessData".GripperCode_R3[3])
      S_Move(in := "AutoProcessData".GripperCode_R3[10], out => "AutoProcessData".GripperCode_R3[4])
   END_RUNG
   RUNG wire#w3
      R_Coil( "ChangeOver_DB".Global.AllFixtureScanCompareOk )
      S_Coil( "ChangeOver_DB".Global.ScanFixtureFlag )
   END_RUNG
   RUNG wire#w1
      Contact( "ChangeOver_DB".Global.ChangeOverRequest )
      wire#w4
      P_Trig( "ChangeOver_DB".P[19] )
      R_Coil( "ChangeOver_DB".Global.AllFixtureScanCompareOk )
   END_RUNG
   RUNG wire#w1
      Contact( "ChangeOver_DB".Global.ScanFixtureFlag )
      Contact( "Station_Sys".Auto.Mode )
   END_RUNG wire#w4
   RUNG wire#w1
      Contact( "ChangeOver_DB".Global.ChangeOverSelected )
   END_RUNG wire#w4
   RUNG wire#w1
      Contact( "ChangeOver_DB".Global.Hmi_ForceChangeOver )
   END_RUNG wire#w4
   // the same network as SCL:
   #_w1 := "AlwaysTRUE" AND ("ChangeOver_DB".Global.ChangeOverRequest OR "ChangeOver_DB".Global.ScanFixtureFlag) AND "Station_Sys".Auto.Mode;
   #_w2 := #_w1 AND NOT "ChangeOver_DB".P[0];   // rising edge
   "ChangeOver_DB".P[0] := #_w1;
   IF #_w2 THEN
       "AutoProcessData".A_Table_1[1] := "AutoProcessData".A_Table_1[10];
       "AutoProcessData".A_Table_1[2] := "AutoProcessData".A_Table_1[10];
       "AutoProcessData".A_Table_1[3] := "AutoProcessData".A_Table_1[10];
       "AutoProcessData".A_Table_1[4] := "AutoProcessData".A_Table_1[10];
       "AutoProcessData".A_Table_1[5] := "AutoProcessData".A_Table_1[10];
       "AutoProcessData".A_Table_1[6] := "AutoProcessData".A_Table_1[10];
       "AutoProcessData".A_Table_1[7] := "AutoProcessData".A_Table_1[10];
       "AutoProcessData".A_Table_1[8] := "AutoProcessData".A_Table_1[10];
       "AutoProcessData".A_Table_2[1] := "AutoProcessData".A_Table_1[10];
       "AutoProcessData".A_Table_2[2] := "AutoProcessData".A_Table_1[10];
       "AutoProcessData".A_Table_2[3] := "AutoProcessData".A_Table_1[10];
       "AutoProcessData".A_Table_2[4] := "AutoProcessData".A_Table_1[10];
       "AutoProcessData".A_Table_2[5] := "AutoProcessData".A_Table_1[10];
       "AutoProcessData".A_Table_2[6] := "AutoProcessData".A_Table_1[10];
       "AutoProcessData".A_Table_2[7] := "AutoProcessData".A_Table_1[10];
       "AutoProcessData".A_Table_2[8] := "AutoProcessData".A_Table_1[10];
       "AutoProcessData".FixtureCode_A1[1] := "AutoProcessData".FixtureCode_A1[10];
       "AutoProcessData".FixtureCode_A1[2] := "AutoProcessData".FixtureCode_A1[10];
       "AutoProcessData".FixtureCode_A1[3] := "AutoProcessData".FixtureCode_A1[10];
       "AutoProcessData".FixtureCode_A1[4] := "AutoProcessData".FixtureCode_A1[10];
       "AutoProcessData".FixtureCode_A1[5] := "AutoProcessData".FixtureCode_A1[10];
       "AutoProcessData".FixtureCode_A1[6] := "AutoProcessData".FixtureCode_A1[10];
       "AutoProcessData".FixtureCode_A1[7] := "AutoProcessData".FixtureCode_A1[10];
       "AutoProcessData".FixtureCode_A2[1] := "AutoProcessData".FixtureCode_A2[10];
       "AutoProcessData".FixtureCode_A2[2] := "AutoProcessData".FixtureCode_A2[10];
       "AutoProcessData".FixtureCode_A2[3] := "AutoProcessData".FixtureCode_A2[10];
       "AutoProcessData".FixtureCode_A2[4] := "AutoProcessData".FixtureCode_A2[10];
       "AutoProcessData".FixtureCode_A2[5] := "AutoProcessData".FixtureCode_A2[10];
       "AutoProcessData".FixtureCode_A2[6] := "AutoProcessData".FixtureCode_A2[10];
       "AutoProcessData".FixtureCode_A2[7] := "AutoProcessData".FixtureCode_A2[10];
       "AutoProcessData".GripperCode_R1[1] := "AutoProcessData".GripperCode_R1[10];
       "AutoProcessData".GripperCode_R1[2] := "AutoProcessData".GripperCode_R1[10];
       "AutoProcessData".GripperCode_R1[3] := "AutoProcessData".GripperCode_R1[10];
       "AutoProcessData".GripperCode_R1[4] := "AutoProcessData".GripperCode_R1[10];
       "AutoProcessData".GripperCode_R2[1] := "AutoProcessData".GripperCode_R2[10];
       "AutoProcessData".GripperCode_R2[2] := "AutoProcessData".GripperCode_R2[10];
       "AutoProcessData".GripperCode_R2[3] := "AutoProcessData".GripperCode_R2[10];
       "AutoProcessData".GripperCode_R2[4] := "AutoProcessData".GripperCode_R2[10];
       "AutoProcessData".GripperCode_R3[1] := "AutoProcessData".GripperCode_R3[10];
       "AutoProcessData".GripperCode_R3[2] := "AutoProcessData".GripperCode_R3[10];
       "AutoProcessData".GripperCode_R3[3] := "AutoProcessData".GripperCode_R3[10];
       "AutoProcessData".GripperCode_R3[4] := "AutoProcessData".GripperCode_R3[10];
       "ChangeOver_DB".Global.AllFixtureScanCompareOk := FALSE;
       "ChangeOver_DB".Global.ScanFixtureFlag := TRUE;
   END_IF;
   #_w3 := "AlwaysTRUE" AND ("ChangeOver_DB".Global.ChangeOverRequest OR ("ChangeOver_DB".Global.ScanFixtureFlag AND "Station_Sys".Auto.Mode) OR "ChangeOver_DB".Global.ChangeOverSelected OR "ChangeOver_DB".Global.Hmi_ForceChangeOver);
   #_w4 := #_w3 AND NOT "ChangeOver_DB".P[19];   // rising edge
   "ChangeOver_DB".P[19] := #_w3;
   IF #_w4 THEN "ChangeOver_DB".Global.AllFixtureScanCompareOk := FALSE; END_IF;
END_REGION

REGION Network 3: ManualModeFlag
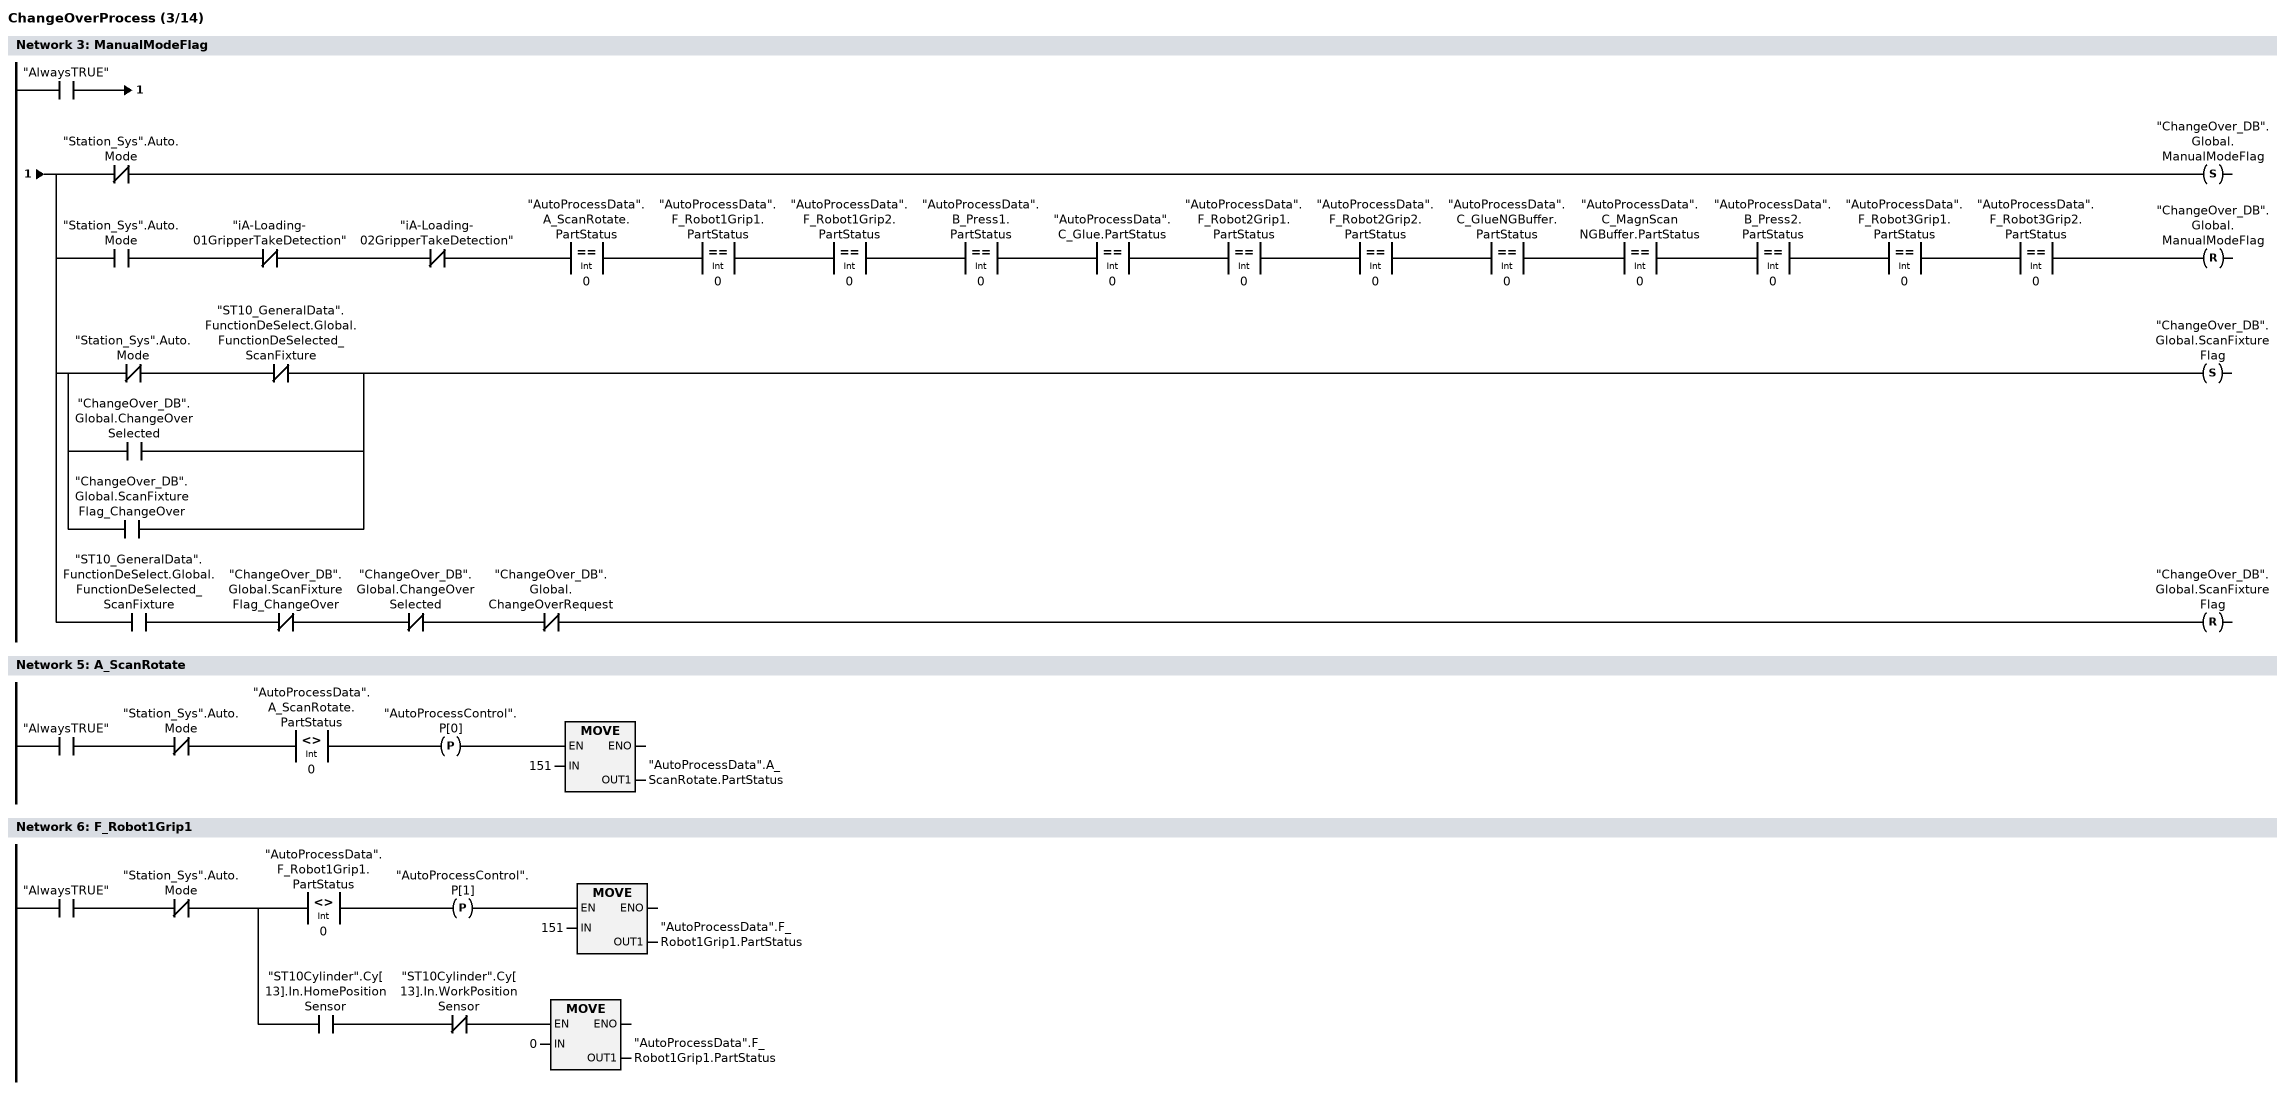
   RUNG wire#powerrail
      Contact( "AlwaysTRUE" )
      wire#w1
      I_Contact( "Station_Sys".Auto.Mode )
      S_Coil( "ChangeOver_DB".Global.ManualModeFlag )
   END_RUNG
   RUNG wire#w1
      Contact( "Station_Sys".Auto.Mode )
      I_Contact( "iA-Loading-01GripperTakeDetection" )
      I_Contact( "iA-Loading-02GripperTakeDetection" )
      { S7_Templates := "SrcType := Int" } EQ_Contact(in1 := "AutoProcessData".A_ScanRotate.PartStatus, in2 := 0)
      { S7_Templates := "SrcType := Int" } EQ_Contact(in1 := "AutoProcessData".F_Robot1Grip1.PartStatus, in2 := 0)
      { S7_Templates := "SrcType := Int" } EQ_Contact(in1 := "AutoProcessData".F_Robot1Grip2.PartStatus, in2 := 0)
      { S7_Templates := "SrcType := Int" } EQ_Contact(in1 := "AutoProcessData".B_Press1.PartStatus, in2 := 0)
      { S7_Templates := "SrcType := Int" } EQ_Contact(in1 := "AutoProcessData".C_Glue.PartStatus, in2 := 0)
      { S7_Templates := "SrcType := Int" } EQ_Contact(in1 := "AutoProcessData".F_Robot2Grip1.PartStatus, in2 := 0)
      { S7_Templates := "SrcType := Int" } EQ_Contact(in1 := "AutoProcessData".F_Robot2Grip2.PartStatus, in2 := 0)
      { S7_Templates := "SrcType := Int" } EQ_Contact(in1 := "AutoProcessData".C_GlueNGBuffer.PartStatus, in2 := 0)
      { S7_Templates := "SrcType := Int" } EQ_Contact(in1 := "AutoProcessData".C_MagnScanNGBuffer.PartStatus, in2 := 0)
      { S7_Templates := "SrcType := Int" } EQ_Contact(in1 := "AutoProcessData".B_Press2.PartStatus, in2 := 0)
      { S7_Templates := "SrcType := Int" } EQ_Contact(in1 := "AutoProcessData".F_Robot3Grip1.PartStatus, in2 := 0)
      { S7_Templates := "SrcType := Int" } EQ_Contact(in1 := "AutoProcessData".F_Robot3Grip2.PartStatus, in2 := 0)
      R_Coil( "ChangeOver_DB".Global.ManualModeFlag )
   END_RUNG
   RUNG wire#w1
      I_Contact( "Station_Sys".Auto.Mode )
      I_Contact( "ST10_GeneralData".FunctionDeSelect.Global.FunctionDeSelected_ScanFixture )
      wire#w2
      S_Coil( "ChangeOver_DB".Global.ScanFixtureFlag )
   END_RUNG
   RUNG wire#w1
      Contact( "ChangeOver_DB".Global.ChangeOverSelected )
   END_RUNG wire#w2
   RUNG wire#w1
      Contact( "ChangeOver_DB".Global.ScanFixtureFlag_ChangeOver )
   END_RUNG wire#w2
   RUNG wire#w1
      Contact( "ST10_GeneralData".FunctionDeSelect.Global.FunctionDeSelected_ScanFixture )
      I_Contact( "ChangeOver_DB".Global.ScanFixtureFlag_ChangeOver )
      I_Contact( "ChangeOver_DB".Global.ChangeOverSelected )
      I_Contact( "ChangeOver_DB".Global.ChangeOverRequest )
      R_Coil( "ChangeOver_DB".Global.ScanFixtureFlag )
   END_RUNG
   // the same network as SCL:
   IF "AlwaysTRUE" AND NOT "Station_Sys".Auto.Mode THEN
       "ChangeOver_DB".Global.ManualModeFlag := TRUE;
   END_IF;
   IF "AlwaysTRUE" AND "Station_Sys".Auto.Mode AND NOT "iA-Loading-01GripperTakeDetection" AND NOT "iA-Loading-02GripperTakeDetection" AND ("AutoProcessData".A_ScanRotate.PartStatus = 0) AND ("AutoProcessData".F_Robot1Grip1.PartStatus = 0) AND ("AutoProcessData".F_Robot1Grip2.PartStatus = 0) AND ("AutoProcessData".B_Press1.PartStatus = 0) AND ("AutoProcessData".C_Glue.PartStatus = 0) AND ("AutoProcessData".F_Robot2Grip1.PartStatus = 0) AND ("AutoProcessData".F_Robot2Grip2.PartStatus = 0) AND ("AutoProcessData".C_GlueNGBuffer.PartStatus = 0) AND ("AutoProcessData".C_MagnScanNGBuffer.PartStatus = 0) AND ("AutoProcessData".B_Press2.PartStatus = 0) AND ("AutoProcessData".F_Robot3Grip1.PartStatus = 0) AND ("AutoProcessData".F_Robot3Grip2.PartStatus = 0) THEN
       "ChangeOver_DB".Global.ManualModeFlag := FALSE;
   END_IF;
   IF "AlwaysTRUE" AND ((NOT "Station_Sys".Auto.Mode AND NOT "ST10_GeneralData".FunctionDeSelect.Global.FunctionDeSelected_ScanFixture) OR "ChangeOver_DB".Global.ChangeOverSelected OR "ChangeOver_DB".Global.ScanFixtureFlag_ChangeOver) THEN
       "ChangeOver_DB".Global.ScanFixtureFlag := TRUE;
   END_IF;
   IF "AlwaysTRUE" AND "ST10_GeneralData".FunctionDeSelect.Global.FunctionDeSelected_ScanFixture AND NOT "ChangeOver_DB".Global.ScanFixtureFlag_ChangeOver AND NOT "ChangeOver_DB".Global.ChangeOverSelected AND NOT "ChangeOver_DB".Global.ChangeOverRequest THEN
       "ChangeOver_DB".Global.ScanFixtureFlag := FALSE;
   END_IF;
END_REGION

REGION Network 4: ----------------------------- Manu Mode,All the part NG -------------------------------------------------------
END_REGION

REGION Network 5: A_ScanRotate
   RUNG wire#powerrail
      Contact( "AlwaysTRUE" )
      I_Contact( "Station_Sys".Auto.Mode )
      { S7_Templates := "SrcType := Int" } NE_Contact(in1 := "AutoProcessData".A_ScanRotate.PartStatus, in2 := 0)
      P_Trig( "AutoProcessControl".P[0] )
      Move(in := 151, out1 => "AutoProcessData".A_ScanRotate.PartStatus)
   END_RUNG
   // the same network as SCL:
   #_w1 := "AlwaysTRUE" AND NOT "Station_Sys".Auto.Mode AND ("AutoProcessData".A_ScanRotate.PartStatus <> 0);
   #_w2 := #_w1 AND NOT "AutoProcessControl".P[0];   // rising edge
   "AutoProcessControl".P[0] := #_w1;
   IF #_w2 THEN "AutoProcessData".A_ScanRotate.PartStatus := 151; END_IF;
END_REGION

REGION Network 6: F_Robot1Grip1
   RUNG wire#powerrail
      Contact( "AlwaysTRUE" )
      I_Contact( "Station_Sys".Auto.Mode )
      wire#w1
      { S7_Templates := "SrcType := Int" } NE_Contact(in1 := "AutoProcessData".F_Robot1Grip1.PartStatus, in2 := 0)
      P_Trig( "AutoProcessControl".P[1] )
      Move(in := 151, out1 => "AutoProcessData".F_Robot1Grip1.PartStatus)
   END_RUNG
   RUNG wire#w1
      Contact( "ST10Cylinder".Cy[13].In.HomePositionSensor )
      I_Contact( "ST10Cylinder".Cy[13].In.WorkPositionSensor )
      Move(in := 0, out1 => "AutoProcessData".F_Robot1Grip1.PartStatus)
   END_RUNG
   // the same network as SCL:
   #_w1 := "AlwaysTRUE" AND NOT "Station_Sys".Auto.Mode;
   #_w2 := #_w1 AND ("AutoProcessData".F_Robot1Grip1.PartStatus <> 0);
   #_w3 := #_w2 AND NOT "AutoProcessControl".P[1];   // rising edge
   "AutoProcessControl".P[1] := #_w2;
   IF #_w3 THEN "AutoProcessData".F_Robot1Grip1.PartStatus := 151; END_IF;
   IF #_w1 AND "ST10Cylinder".Cy[13].In.HomePositionSensor AND NOT "ST10Cylinder".Cy[13].In.WorkPositionSensor THEN
       "AutoProcessData".F_Robot1Grip1.PartStatus := 0;
   END_IF;
END_REGION

REGION Network 7: F_Robot1Grip2
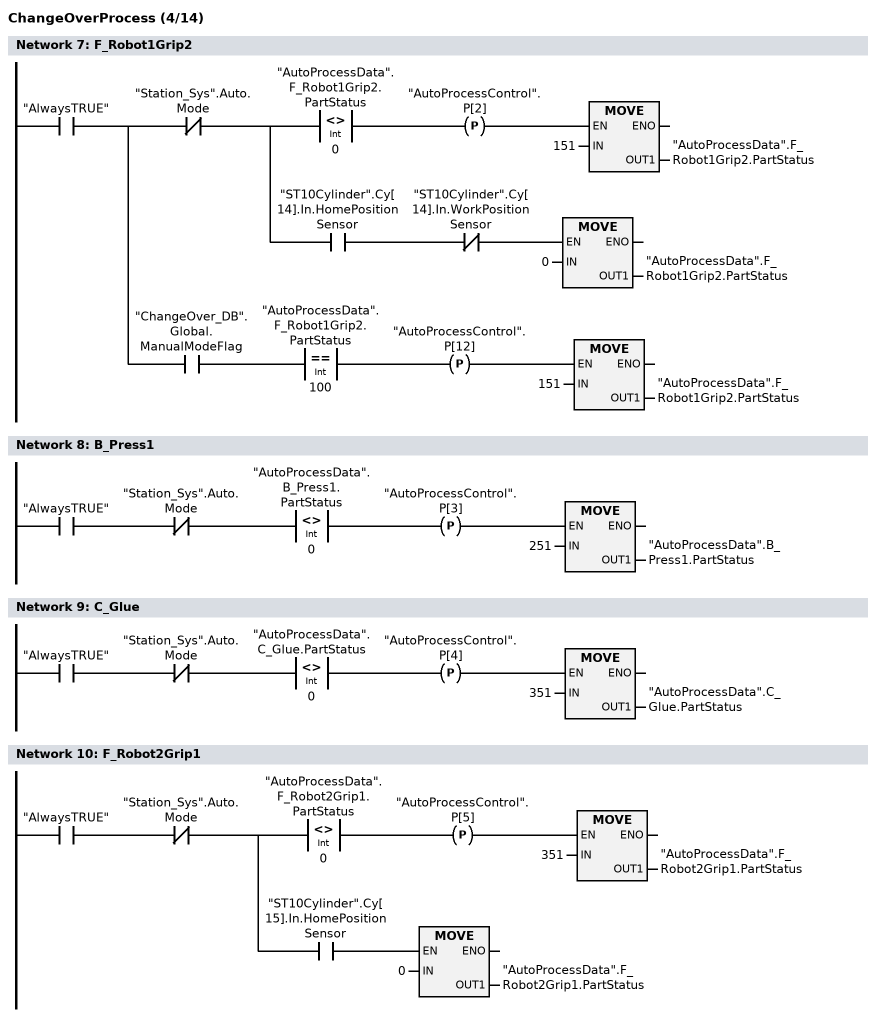
   RUNG wire#powerrail
      Contact( "AlwaysTRUE" )
      wire#w1
      I_Contact( "Station_Sys".Auto.Mode )
      wire#w2
      { S7_Templates := "SrcType := Int" } NE_Contact(in1 := "AutoProcessData".F_Robot1Grip2.PartStatus, in2 := 0)
      P_Trig( "AutoProcessControl".P[2] )
      Move(in := 151, out1 => "AutoProcessData".F_Robot1Grip2.PartStatus)
   END_RUNG
   RUNG wire#w2
      Contact( "ST10Cylinder".Cy[14].In.HomePositionSensor )
      I_Contact( "ST10Cylinder".Cy[14].In.WorkPositionSensor )
      Move(in := 0, out1 => "AutoProcessData".F_Robot1Grip2.PartStatus)
   END_RUNG
   RUNG wire#w1
      Contact( "ChangeOver_DB".Global.ManualModeFlag )
      { S7_Templates := "SrcType := Int" } EQ_Contact(in1 := "AutoProcessData".F_Robot1Grip2.PartStatus, in2 := 100)
      P_Trig( "AutoProcessControl".P[12] )
      Move(in := 151, out1 => "AutoProcessData".F_Robot1Grip2.PartStatus)
   END_RUNG
   // the same network as SCL:
   #_w1 := "AlwaysTRUE" AND NOT "Station_Sys".Auto.Mode;
   #_w2 := #_w1 AND ("AutoProcessData".F_Robot1Grip2.PartStatus <> 0);
   #_w3 := #_w2 AND NOT "AutoProcessControl".P[2];   // rising edge
   "AutoProcessControl".P[2] := #_w2;
   IF #_w3 THEN "AutoProcessData".F_Robot1Grip2.PartStatus := 151; END_IF;
   IF #_w1 AND "ST10Cylinder".Cy[14].In.HomePositionSensor AND NOT "ST10Cylinder".Cy[14].In.WorkPositionSensor THEN
       "AutoProcessData".F_Robot1Grip2.PartStatus := 0;
   END_IF;
   #_w4 := "AlwaysTRUE" AND "ChangeOver_DB".Global.ManualModeFlag AND ("AutoProcessData".F_Robot1Grip2.PartStatus = 100);
   #_w5 := #_w4 AND NOT "AutoProcessControl".P[12];   // rising edge
   "AutoProcessControl".P[12] := #_w4;
   IF #_w5 THEN "AutoProcessData".F_Robot1Grip2.PartStatus := 151; END_IF;
END_REGION

REGION Network 8: B_Press1
   RUNG wire#powerrail
      Contact( "AlwaysTRUE" )
      I_Contact( "Station_Sys".Auto.Mode )
      { S7_Templates := "SrcType := Int" } NE_Contact(in1 := "AutoProcessData".B_Press1.PartStatus, in2 := 0)
      P_Trig( "AutoProcessControl".P[3] )
      Move(in := 251, out1 => "AutoProcessData".B_Press1.PartStatus)
   END_RUNG
   // the same network as SCL:
   #_w1 := "AlwaysTRUE" AND NOT "Station_Sys".Auto.Mode AND ("AutoProcessData".B_Press1.PartStatus <> 0);
   #_w2 := #_w1 AND NOT "AutoProcessControl".P[3];   // rising edge
   "AutoProcessControl".P[3] := #_w1;
   IF #_w2 THEN "AutoProcessData".B_Press1.PartStatus := 251; END_IF;
END_REGION

REGION Network 9: C_Glue
   RUNG wire#powerrail
      Contact( "AlwaysTRUE" )
      I_Contact( "Station_Sys".Auto.Mode )
      { S7_Templates := "SrcType := Int" } NE_Contact(in1 := "AutoProcessData".C_Glue.PartStatus, in2 := 0)
      P_Trig( "AutoProcessControl".P[4] )
      Move(in := 351, out1 => "AutoProcessData".C_Glue.PartStatus)
   END_RUNG
   // the same network as SCL:
   #_w1 := "AlwaysTRUE" AND NOT "Station_Sys".Auto.Mode AND ("AutoProcessData".C_Glue.PartStatus <> 0);
   #_w2 := #_w1 AND NOT "AutoProcessControl".P[4];   // rising edge
   "AutoProcessControl".P[4] := #_w1;
   IF #_w2 THEN "AutoProcessData".C_Glue.PartStatus := 351; END_IF;
END_REGION

REGION Network 10: F_Robot2Grip1
   RUNG wire#powerrail
      Contact( "AlwaysTRUE" )
      I_Contact( "Station_Sys".Auto.Mode )
      wire#w1
      { S7_Templates := "SrcType := Int" } NE_Contact(in1 := "AutoProcessData".F_Robot2Grip1.PartStatus, in2 := 0)
      P_Trig( "AutoProcessControl".P[5] )
      Move(in := 351, out1 => "AutoProcessData".F_Robot2Grip1.PartStatus)
   END_RUNG
   RUNG wire#w1
      Contact( "ST10Cylinder".Cy[15].In.HomePositionSensor )
      Move(in := 0, out1 => "AutoProcessData".F_Robot2Grip1.PartStatus)
   END_RUNG
   // the same network as SCL:
   #_w1 := "AlwaysTRUE" AND NOT "Station_Sys".Auto.Mode;
   #_w2 := #_w1 AND ("AutoProcessData".F_Robot2Grip1.PartStatus <> 0);
   #_w3 := #_w2 AND NOT "AutoProcessControl".P[5];   // rising edge
   "AutoProcessControl".P[5] := #_w2;
   IF #_w3 THEN "AutoProcessData".F_Robot2Grip1.PartStatus := 351; END_IF;
   IF #_w1 AND "ST10Cylinder".Cy[15].In.HomePositionSensor THEN
       "AutoProcessData".F_Robot2Grip1.PartStatus := 0;
   END_IF;
END_REGION

REGION Network 11: F_Robot2Grip2
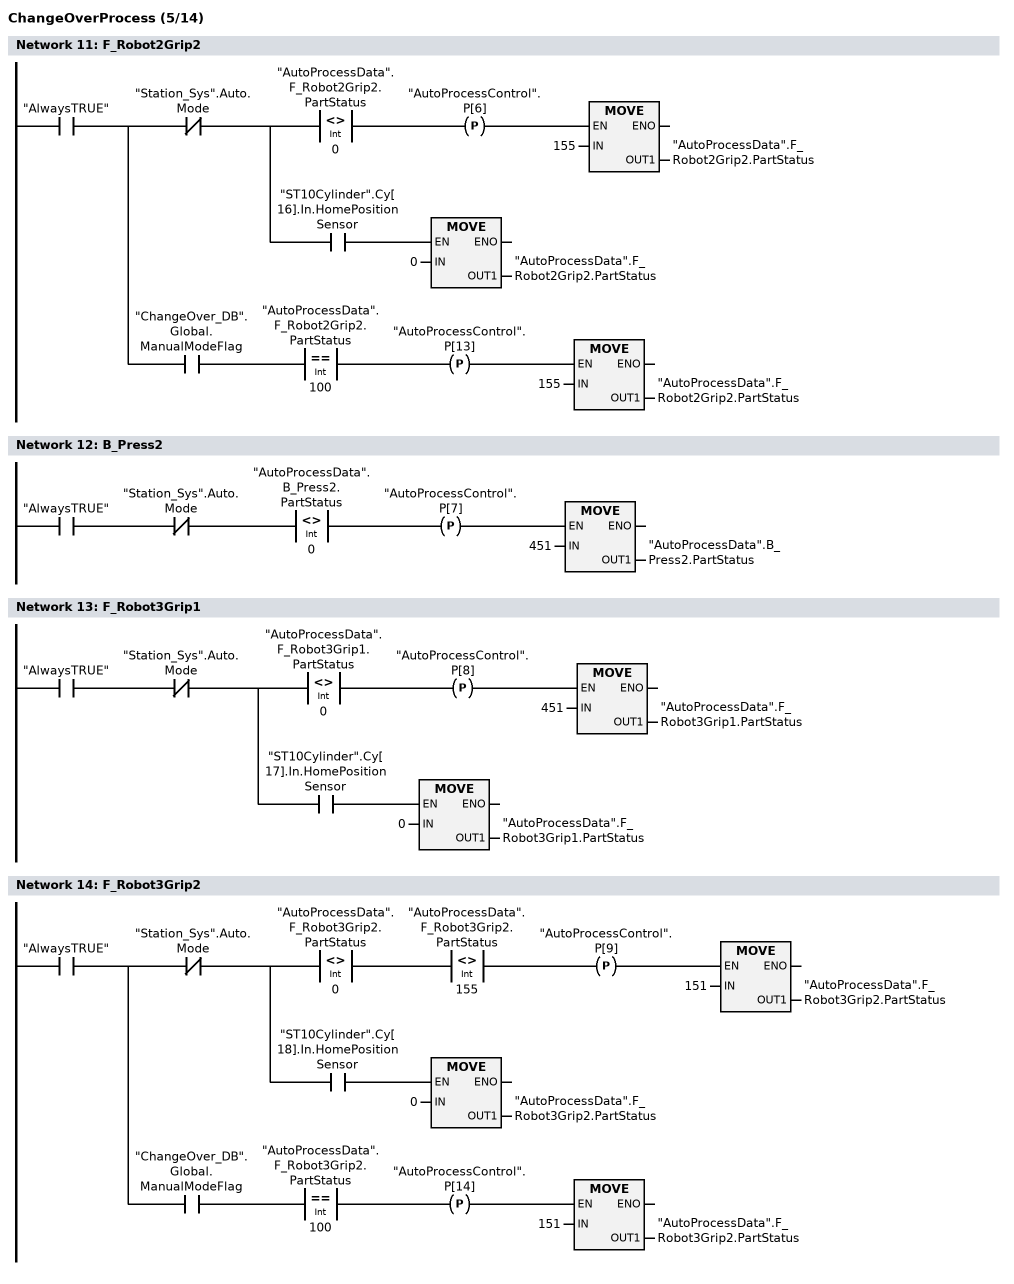
   RUNG wire#powerrail
      Contact( "AlwaysTRUE" )
      wire#w1
      I_Contact( "Station_Sys".Auto.Mode )
      wire#w2
      { S7_Templates := "SrcType := Int" } NE_Contact(in1 := "AutoProcessData".F_Robot2Grip2.PartStatus, in2 := 0)
      P_Trig( "AutoProcessControl".P[6] )
      Move(in := 155, out1 => "AutoProcessData".F_Robot2Grip2.PartStatus)
   END_RUNG
   RUNG wire#w2
      Contact( "ST10Cylinder".Cy[16].In.HomePositionSensor )
      Move(in := 0, out1 => "AutoProcessData".F_Robot2Grip2.PartStatus)
   END_RUNG
   RUNG wire#w1
      Contact( "ChangeOver_DB".Global.ManualModeFlag )
      { S7_Templates := "SrcType := Int" } EQ_Contact(in1 := "AutoProcessData".F_Robot2Grip2.PartStatus, in2 := 100)
      P_Trig( "AutoProcessControl".P[13] )
      Move(in := 155, out1 => "AutoProcessData".F_Robot2Grip2.PartStatus)
   END_RUNG
   // the same network as SCL:
   #_w1 := "AlwaysTRUE" AND NOT "Station_Sys".Auto.Mode;
   #_w2 := #_w1 AND ("AutoProcessData".F_Robot2Grip2.PartStatus <> 0);
   #_w3 := #_w2 AND NOT "AutoProcessControl".P[6];   // rising edge
   "AutoProcessControl".P[6] := #_w2;
   IF #_w3 THEN "AutoProcessData".F_Robot2Grip2.PartStatus := 155; END_IF;
   IF #_w1 AND "ST10Cylinder".Cy[16].In.HomePositionSensor THEN
       "AutoProcessData".F_Robot2Grip2.PartStatus := 0;
   END_IF;
   #_w4 := "AlwaysTRUE" AND "ChangeOver_DB".Global.ManualModeFlag AND ("AutoProcessData".F_Robot2Grip2.PartStatus = 100);
   #_w5 := #_w4 AND NOT "AutoProcessControl".P[13];   // rising edge
   "AutoProcessControl".P[13] := #_w4;
   IF #_w5 THEN "AutoProcessData".F_Robot2Grip2.PartStatus := 155; END_IF;
END_REGION

REGION Network 12: B_Press2
   RUNG wire#powerrail
      Contact( "AlwaysTRUE" )
      I_Contact( "Station_Sys".Auto.Mode )
      { S7_Templates := "SrcType := Int" } NE_Contact(in1 := "AutoProcessData".B_Press2.PartStatus, in2 := 0)
      P_Trig( "AutoProcessControl".P[7] )
      Move(in := 451, out1 => "AutoProcessData".B_Press2.PartStatus)
   END_RUNG
   // the same network as SCL:
   #_w1 := "AlwaysTRUE" AND NOT "Station_Sys".Auto.Mode AND ("AutoProcessData".B_Press2.PartStatus <> 0);
   #_w2 := #_w1 AND NOT "AutoProcessControl".P[7];   // rising edge
   "AutoProcessControl".P[7] := #_w1;
   IF #_w2 THEN "AutoProcessData".B_Press2.PartStatus := 451; END_IF;
END_REGION

REGION Network 13: F_Robot3Grip1
   RUNG wire#powerrail
      Contact( "AlwaysTRUE" )
      I_Contact( "Station_Sys".Auto.Mode )
      wire#w1
      { S7_Templates := "SrcType := Int" } NE_Contact(in1 := "AutoProcessData".F_Robot3Grip1.PartStatus, in2 := 0)
      P_Trig( "AutoProcessControl".P[8] )
      Move(in := 451, out1 => "AutoProcessData".F_Robot3Grip1.PartStatus)
   END_RUNG
   RUNG wire#w1
      Contact( "ST10Cylinder".Cy[17].In.HomePositionSensor )
      Move(in := 0, out1 => "AutoProcessData".F_Robot3Grip1.PartStatus)
   END_RUNG
   // the same network as SCL:
   #_w1 := "AlwaysTRUE" AND NOT "Station_Sys".Auto.Mode;
   #_w2 := #_w1 AND ("AutoProcessData".F_Robot3Grip1.PartStatus <> 0);
   #_w3 := #_w2 AND NOT "AutoProcessControl".P[8];   // rising edge
   "AutoProcessControl".P[8] := #_w2;
   IF #_w3 THEN "AutoProcessData".F_Robot3Grip1.PartStatus := 451; END_IF;
   IF #_w1 AND "ST10Cylinder".Cy[17].In.HomePositionSensor THEN
       "AutoProcessData".F_Robot3Grip1.PartStatus := 0;
   END_IF;
END_REGION

REGION Network 14: F_Robot3Grip2
   RUNG wire#powerrail
      Contact( "AlwaysTRUE" )
      wire#w1
      I_Contact( "Station_Sys".Auto.Mode )
      wire#w2
      { S7_Templates := "SrcType := Int" } NE_Contact(in1 := "AutoProcessData".F_Robot3Grip2.PartStatus, in2 := 0)
      { S7_Templates := "SrcType := Int" } NE_Contact(in1 := "AutoProcessData".F_Robot3Grip2.PartStatus, in2 := 155)
      P_Trig( "AutoProcessControl".P[9] )
      Move(in := 151, out1 => "AutoProcessData".F_Robot3Grip2.PartStatus)
   END_RUNG
   RUNG wire#w2
      Contact( "ST10Cylinder".Cy[18].In.HomePositionSensor )
      Move(in := 0, out1 => "AutoProcessData".F_Robot3Grip2.PartStatus)
   END_RUNG
   RUNG wire#w1
      Contact( "ChangeOver_DB".Global.ManualModeFlag )
      { S7_Templates := "SrcType := Int" } EQ_Contact(in1 := "AutoProcessData".F_Robot3Grip2.PartStatus, in2 := 100)
      P_Trig( "AutoProcessControl".P[14] )
      Move(in := 151, out1 => "AutoProcessData".F_Robot3Grip2.PartStatus)
   END_RUNG
   // the same network as SCL:
   #_w1 := "AlwaysTRUE" AND NOT "Station_Sys".Auto.Mode;
   #_w2 := #_w1 AND ("AutoProcessData".F_Robot3Grip2.PartStatus <> 0) AND ("AutoProcessData".F_Robot3Grip2.PartStatus <> 155);
   #_w3 := #_w2 AND NOT "AutoProcessControl".P[9];   // rising edge
   "AutoProcessControl".P[9] := #_w2;
   IF #_w3 THEN "AutoProcessData".F_Robot3Grip2.PartStatus := 151; END_IF;
   IF #_w1 AND "ST10Cylinder".Cy[18].In.HomePositionSensor THEN
       "AutoProcessData".F_Robot3Grip2.PartStatus := 0;
   END_IF;
   #_w4 := "AlwaysTRUE" AND "ChangeOver_DB".Global.ManualModeFlag AND ("AutoProcessData".F_Robot3Grip2.PartStatus = 100);
   #_w5 := #_w4 AND NOT "AutoProcessControl".P[14];   // rising edge
   "AutoProcessControl".P[14] := #_w4;
   IF #_w5 THEN "AutoProcessData".F_Robot3Grip2.PartStatus := 151; END_IF;
END_REGION

REGION Network 15: ---------------------------------- FixtureCode ------------------------------------------
END_REGION

REGION Network 16: A1_Table
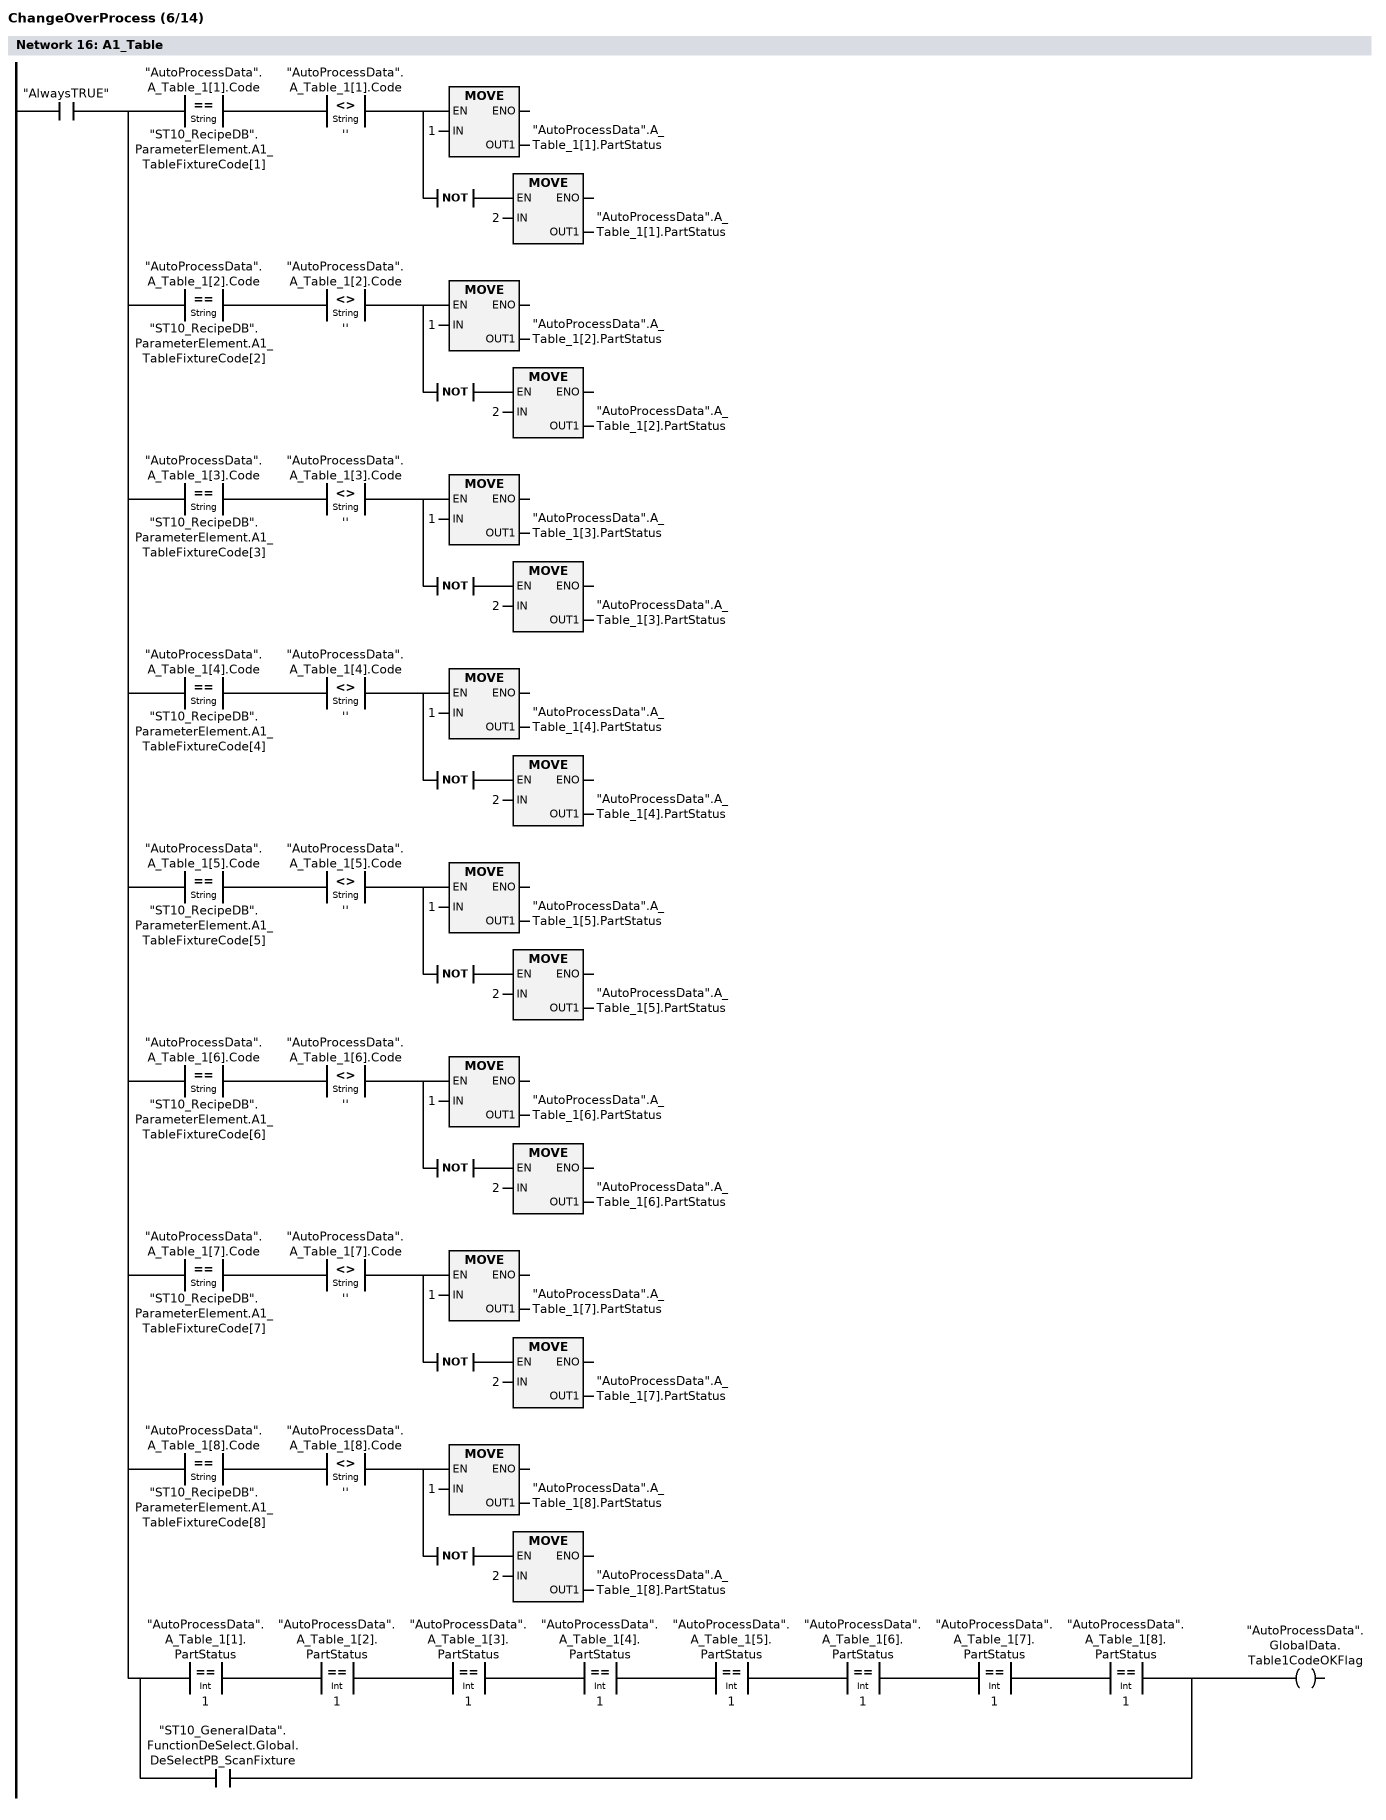
   RUNG wire#powerrail
      Contact( "AlwaysTRUE" )
      wire#w1
      { S7_Templates := "SrcType := String" } EQ_Contact(in1 := "AutoProcessData".A_Table_1[1].Code, in2 := "ST10_RecipeDB".ParameterElement.A1_TableFixtureCode[1])
      { S7_Templates := "SrcType := String" } NE_Contact(in1 := "AutoProcessData".A_Table_1[1].Code, in2 := '')
      wire#w2
      Move(in := 1, out1 => "AutoProcessData".A_Table_1[1].PartStatus)
   END_RUNG
   RUNG wire#w2
      Not()
      Move(in := 2, out1 => "AutoProcessData".A_Table_1[1].PartStatus)
   END_RUNG
   RUNG wire#w1
      { S7_Templates := "SrcType := String" } EQ_Contact(in1 := "AutoProcessData".A_Table_1[2].Code, in2 := "ST10_RecipeDB".ParameterElement.A1_TableFixtureCode[2])
      { S7_Templates := "SrcType := String" } NE_Contact(in1 := "AutoProcessData".A_Table_1[2].Code, in2 := '')
      wire#w3
      Move(in := 1, out1 => "AutoProcessData".A_Table_1[2].PartStatus)
   END_RUNG
   RUNG wire#w3
      Not()
      Move(in := 2, out1 => "AutoProcessData".A_Table_1[2].PartStatus)
   END_RUNG
   RUNG wire#w1
      { S7_Templates := "SrcType := String" } EQ_Contact(in1 := "AutoProcessData".A_Table_1[3].Code, in2 := "ST10_RecipeDB".ParameterElement.A1_TableFixtureCode[3])
      { S7_Templates := "SrcType := String" } NE_Contact(in1 := "AutoProcessData".A_Table_1[3].Code, in2 := '')
      wire#w4
      Move(in := 1, out1 => "AutoProcessData".A_Table_1[3].PartStatus)
   END_RUNG
   RUNG wire#w4
      Not()
      Move(in := 2, out1 => "AutoProcessData".A_Table_1[3].PartStatus)
   END_RUNG
   RUNG wire#w1
      { S7_Templates := "SrcType := String" } EQ_Contact(in1 := "AutoProcessData".A_Table_1[4].Code, in2 := "ST10_RecipeDB".ParameterElement.A1_TableFixtureCode[4])
      { S7_Templates := "SrcType := String" } NE_Contact(in1 := "AutoProcessData".A_Table_1[4].Code, in2 := '')
      wire#w5
      Move(in := 1, out1 => "AutoProcessData".A_Table_1[4].PartStatus)
   END_RUNG
   RUNG wire#w5
      Not()
      Move(in := 2, out1 => "AutoProcessData".A_Table_1[4].PartStatus)
   END_RUNG
   RUNG wire#w1
      { S7_Templates := "SrcType := String" } EQ_Contact(in1 := "AutoProcessData".A_Table_1[5].Code, in2 := "ST10_RecipeDB".ParameterElement.A1_TableFixtureCode[5])
      { S7_Templates := "SrcType := String" } NE_Contact(in1 := "AutoProcessData".A_Table_1[5].Code, in2 := '')
      wire#w6
      Move(in := 1, out1 => "AutoProcessData".A_Table_1[5].PartStatus)
   END_RUNG
   RUNG wire#w6
      Not()
      Move(in := 2, out1 => "AutoProcessData".A_Table_1[5].PartStatus)
   END_RUNG
   RUNG wire#w1
      { S7_Templates := "SrcType := String" } EQ_Contact(in1 := "AutoProcessData".A_Table_1[6].Code, in2 := "ST10_RecipeDB".ParameterElement.A1_TableFixtureCode[6])
      { S7_Templates := "SrcType := String" } NE_Contact(in1 := "AutoProcessData".A_Table_1[6].Code, in2 := '')
      wire#w7
      Move(in := 1, out1 => "AutoProcessData".A_Table_1[6].PartStatus)
   END_RUNG
   RUNG wire#w7
      Not()
      Move(in := 2, out1 => "AutoProcessData".A_Table_1[6].PartStatus)
   END_RUNG
   RUNG wire#w1
      { S7_Templates := "SrcType := String" } EQ_Contact(in1 := "AutoProcessData".A_Table_1[7].Code, in2 := "ST10_RecipeDB".ParameterElement.A1_TableFixtureCode[7])
      { S7_Templates := "SrcType := String" } NE_Contact(in1 := "AutoProcessData".A_Table_1[7].Code, in2 := '')
      wire#w8
      Move(in := 1, out1 => "AutoProcessData".A_Table_1[7].PartStatus)
   END_RUNG
   RUNG wire#w8
      Not()
      Move(in := 2, out1 => "AutoProcessData".A_Table_1[7].PartStatus)
   END_RUNG
   RUNG wire#w1
      { S7_Templates := "SrcType := String" } EQ_Contact(in1 := "AutoProcessData".A_Table_1[8].Code, in2 := "ST10_RecipeDB".ParameterElement.A1_TableFixtureCode[8])
      { S7_Templates := "SrcType := String" } NE_Contact(in1 := "AutoProcessData".A_Table_1[8].Code, in2 := '')
      wire#w9
      Move(in := 1, out1 => "AutoProcessData".A_Table_1[8].PartStatus)
   END_RUNG
   RUNG wire#w9
      Not()
      Move(in := 2, out1 => "AutoProcessData".A_Table_1[8].PartStatus)
   END_RUNG
   RUNG wire#w1
      { S7_Templates := "SrcType := Int" } EQ_Contact(in1 := "AutoProcessData".A_Table_1[1].PartStatus, in2 := 1)
      { S7_Templates := "SrcType := Int" } EQ_Contact(in1 := "AutoProcessData".A_Table_1[2].PartStatus, in2 := 1)
      { S7_Templates := "SrcType := Int" } EQ_Contact(in1 := "AutoProcessData".A_Table_1[3].PartStatus, in2 := 1)
      { S7_Templates := "SrcType := Int" } EQ_Contact(in1 := "AutoProcessData".A_Table_1[4].PartStatus, in2 := 1)
      { S7_Templates := "SrcType := Int" } EQ_Contact(in1 := "AutoProcessData".A_Table_1[5].PartStatus, in2 := 1)
      { S7_Templates := "SrcType := Int" } EQ_Contact(in1 := "AutoProcessData".A_Table_1[6].PartStatus, in2 := 1)
      { S7_Templates := "SrcType := Int" } EQ_Contact(in1 := "AutoProcessData".A_Table_1[7].PartStatus, in2 := 1)
      { S7_Templates := "SrcType := Int" } EQ_Contact(in1 := "AutoProcessData".A_Table_1[8].PartStatus, in2 := 1)
      wire#w10
      Coil( "AutoProcessData".GlobalData.Table1CodeOKFlag )
   END_RUNG
   RUNG wire#w1
      Contact( "ST10_GeneralData".FunctionDeSelect.Global.DeSelectPB_ScanFixture )
   END_RUNG wire#w10
   // the same network as SCL:
   #_w1 := "AlwaysTRUE" AND ("AutoProcessData".A_Table_1[1].Code = "ST10_RecipeDB".ParameterElement.A1_TableFixtureCode[1]) AND ("AutoProcessData".A_Table_1[1].Code <> '');
   IF #_w1 THEN "AutoProcessData".A_Table_1[1].PartStatus := 1; END_IF;
   IF NOT #_w1 THEN "AutoProcessData".A_Table_1[1].PartStatus := 2; END_IF;
   #_w2 := "AlwaysTRUE" AND ("AutoProcessData".A_Table_1[2].Code = "ST10_RecipeDB".ParameterElement.A1_TableFixtureCode[2]) AND ("AutoProcessData".A_Table_1[2].Code <> '');
   IF #_w2 THEN "AutoProcessData".A_Table_1[2].PartStatus := 1; END_IF;
   IF NOT #_w2 THEN "AutoProcessData".A_Table_1[2].PartStatus := 2; END_IF;
   #_w3 := "AlwaysTRUE" AND ("AutoProcessData".A_Table_1[3].Code = "ST10_RecipeDB".ParameterElement.A1_TableFixtureCode[3]) AND ("AutoProcessData".A_Table_1[3].Code <> '');
   IF #_w3 THEN "AutoProcessData".A_Table_1[3].PartStatus := 1; END_IF;
   IF NOT #_w3 THEN "AutoProcessData".A_Table_1[3].PartStatus := 2; END_IF;
   #_w4 := "AlwaysTRUE" AND ("AutoProcessData".A_Table_1[4].Code = "ST10_RecipeDB".ParameterElement.A1_TableFixtureCode[4]) AND ("AutoProcessData".A_Table_1[4].Code <> '');
   IF #_w4 THEN "AutoProcessData".A_Table_1[4].PartStatus := 1; END_IF;
   IF NOT #_w4 THEN "AutoProcessData".A_Table_1[4].PartStatus := 2; END_IF;
   #_w5 := "AlwaysTRUE" AND ("AutoProcessData".A_Table_1[5].Code = "ST10_RecipeDB".ParameterElement.A1_TableFixtureCode[5]) AND ("AutoProcessData".A_Table_1[5].Code <> '');
   IF #_w5 THEN "AutoProcessData".A_Table_1[5].PartStatus := 1; END_IF;
   IF NOT #_w5 THEN "AutoProcessData".A_Table_1[5].PartStatus := 2; END_IF;
   #_w6 := "AlwaysTRUE" AND ("AutoProcessData".A_Table_1[6].Code = "ST10_RecipeDB".ParameterElement.A1_TableFixtureCode[6]) AND ("AutoProcessData".A_Table_1[6].Code <> '');
   IF #_w6 THEN "AutoProcessData".A_Table_1[6].PartStatus := 1; END_IF;
   IF NOT #_w6 THEN "AutoProcessData".A_Table_1[6].PartStatus := 2; END_IF;
   #_w7 := "AlwaysTRUE" AND ("AutoProcessData".A_Table_1[7].Code = "ST10_RecipeDB".ParameterElement.A1_TableFixtureCode[7]) AND ("AutoProcessData".A_Table_1[7].Code <> '');
   IF #_w7 THEN "AutoProcessData".A_Table_1[7].PartStatus := 1; END_IF;
   IF NOT #_w7 THEN "AutoProcessData".A_Table_1[7].PartStatus := 2; END_IF;
   #_w8 := "AlwaysTRUE" AND ("AutoProcessData".A_Table_1[8].Code = "ST10_RecipeDB".ParameterElement.A1_TableFixtureCode[8]) AND ("AutoProcessData".A_Table_1[8].Code <> '');
   IF #_w8 THEN "AutoProcessData".A_Table_1[8].PartStatus := 1; END_IF;
   IF NOT #_w8 THEN "AutoProcessData".A_Table_1[8].PartStatus := 2; END_IF;
   "AutoProcessData".GlobalData.Table1CodeOKFlag := "AlwaysTRUE" AND ((("AutoProcessData".A_Table_1[1].PartStatus = 1) AND ("AutoProcessData".A_Table_1[2].PartStatus = 1) AND ("AutoProcessData".A_Table_1[3].PartStatus = 1) AND ("AutoProcessData".A_Table_1[4].PartStatus = 1) AND ("AutoProcessData".A_Table_1[5].PartStatus = 1) AND ("AutoProcessData".A_Table_1[6].PartStatus = 1) AND ("AutoProcessData".A_Table_1[7].PartStatus = 1) AND ("AutoProcessData".A_Table_1[8].PartStatus = 1)) OR "ST10_GeneralData".FunctionDeSelect.Global.DeSelectPB_ScanFixture);
END_REGION

REGION Network 17: A2_Table
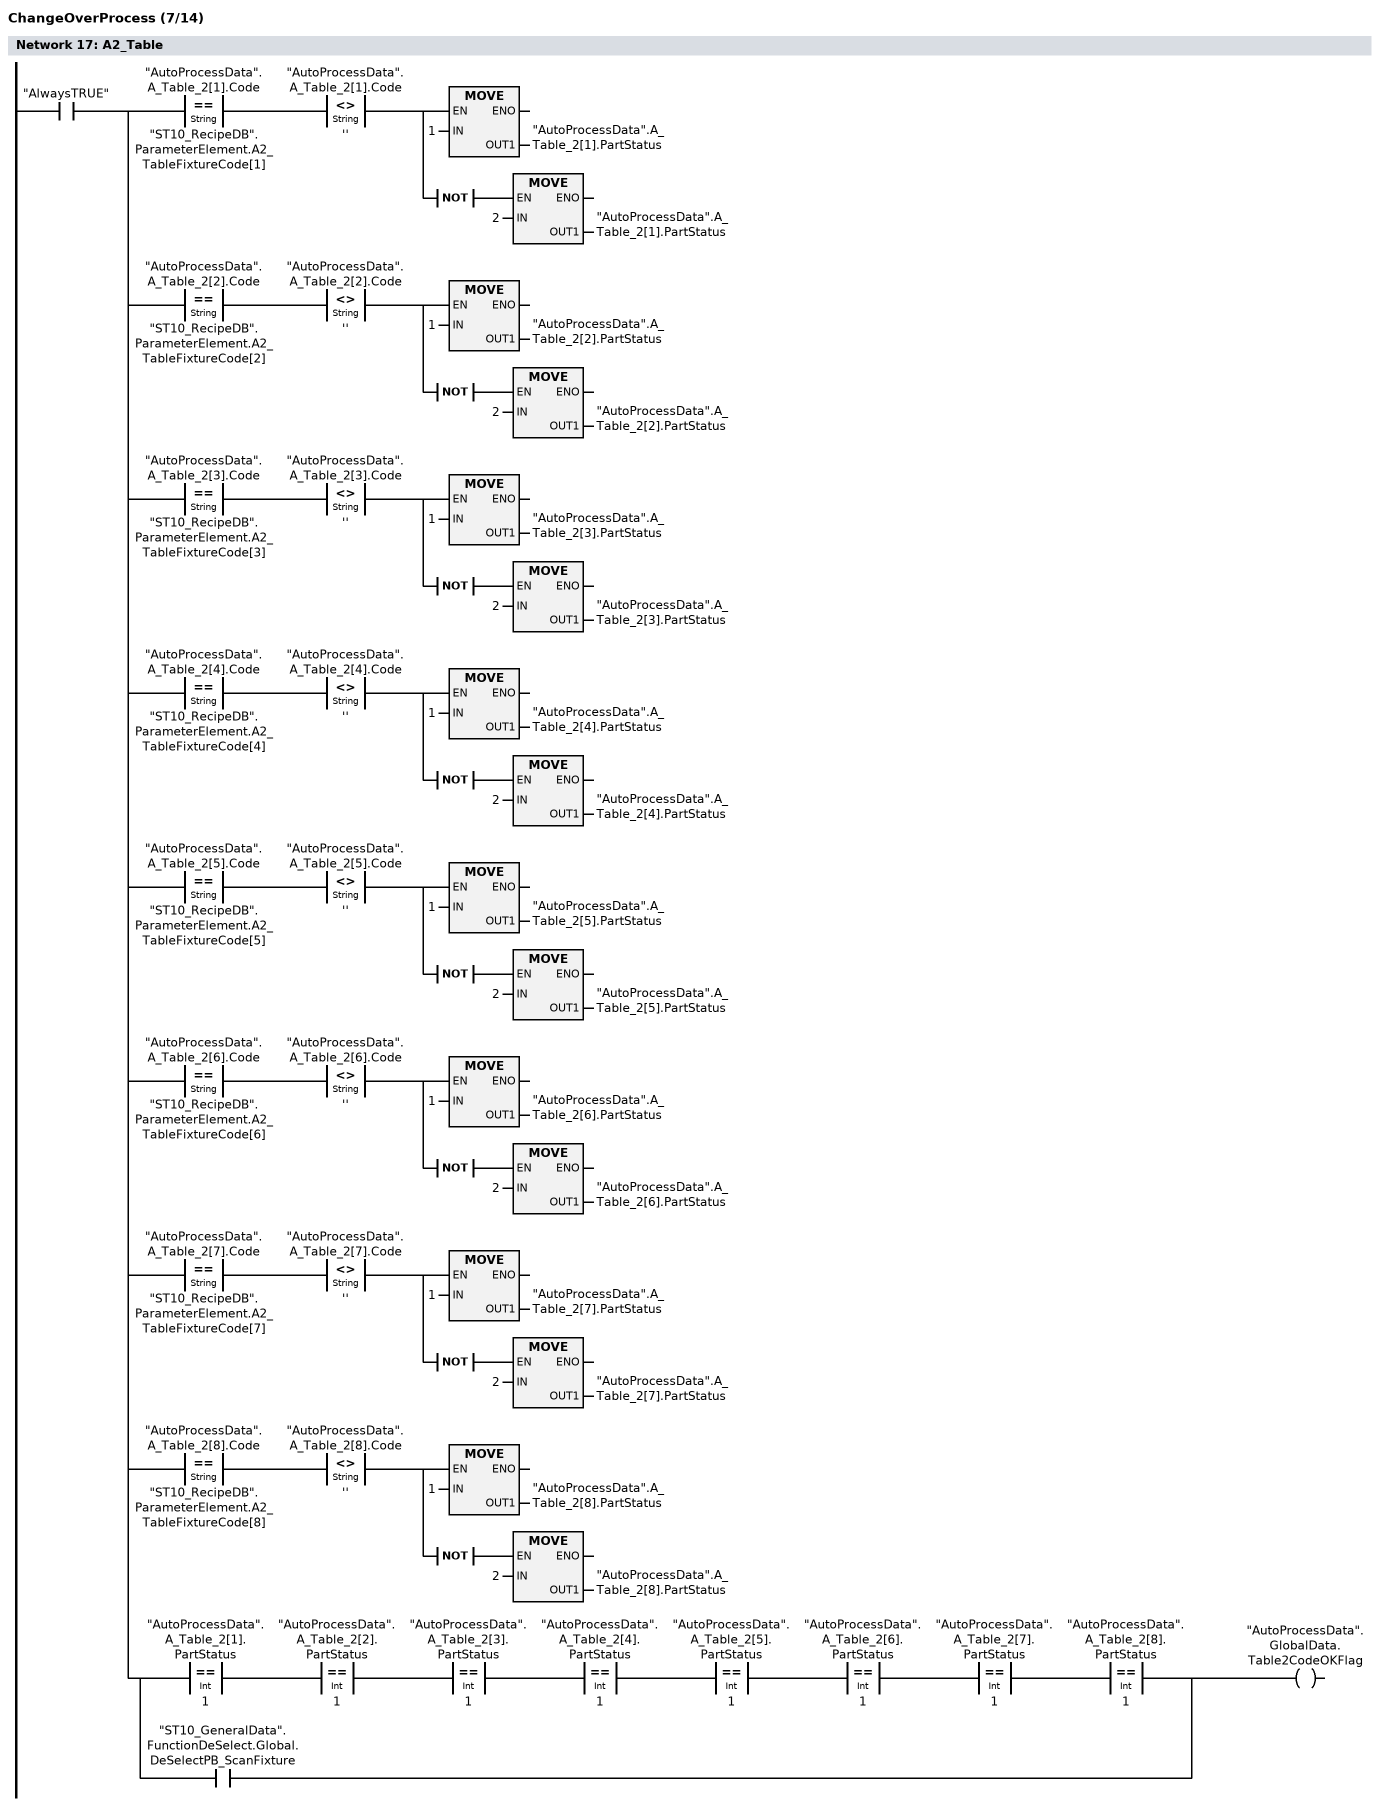
   RUNG wire#powerrail
      Contact( "AlwaysTRUE" )
      wire#w1
      { S7_Templates := "SrcType := String" } EQ_Contact(in1 := "AutoProcessData".A_Table_2[1].Code, in2 := "ST10_RecipeDB".ParameterElement.A2_TableFixtureCode[1])
      { S7_Templates := "SrcType := String" } NE_Contact(in1 := "AutoProcessData".A_Table_2[1].Code, in2 := '')
      wire#w2
      Move(in := 1, out1 => "AutoProcessData".A_Table_2[1].PartStatus)
   END_RUNG
   RUNG wire#w2
      Not()
      Move(in := 2, out1 => "AutoProcessData".A_Table_2[1].PartStatus)
   END_RUNG
   RUNG wire#w1
      { S7_Templates := "SrcType := String" } EQ_Contact(in1 := "AutoProcessData".A_Table_2[2].Code, in2 := "ST10_RecipeDB".ParameterElement.A2_TableFixtureCode[2])
      { S7_Templates := "SrcType := String" } NE_Contact(in1 := "AutoProcessData".A_Table_2[2].Code, in2 := '')
      wire#w3
      Move(in := 1, out1 => "AutoProcessData".A_Table_2[2].PartStatus)
   END_RUNG
   RUNG wire#w3
      Not()
      Move(in := 2, out1 => "AutoProcessData".A_Table_2[2].PartStatus)
   END_RUNG
   RUNG wire#w1
      { S7_Templates := "SrcType := String" } EQ_Contact(in1 := "AutoProcessData".A_Table_2[3].Code, in2 := "ST10_RecipeDB".ParameterElement.A2_TableFixtureCode[3])
      { S7_Templates := "SrcType := String" } NE_Contact(in1 := "AutoProcessData".A_Table_2[3].Code, in2 := '')
      wire#w4
      Move(in := 1, out1 => "AutoProcessData".A_Table_2[3].PartStatus)
   END_RUNG
   RUNG wire#w4
      Not()
      Move(in := 2, out1 => "AutoProcessData".A_Table_2[3].PartStatus)
   END_RUNG
   RUNG wire#w1
      { S7_Templates := "SrcType := String" } EQ_Contact(in1 := "AutoProcessData".A_Table_2[4].Code, in2 := "ST10_RecipeDB".ParameterElement.A2_TableFixtureCode[4])
      { S7_Templates := "SrcType := String" } NE_Contact(in1 := "AutoProcessData".A_Table_2[4].Code, in2 := '')
      wire#w5
      Move(in := 1, out1 => "AutoProcessData".A_Table_2[4].PartStatus)
   END_RUNG
   RUNG wire#w5
      Not()
      Move(in := 2, out1 => "AutoProcessData".A_Table_2[4].PartStatus)
   END_RUNG
   RUNG wire#w1
      { S7_Templates := "SrcType := String" } EQ_Contact(in1 := "AutoProcessData".A_Table_2[5].Code, in2 := "ST10_RecipeDB".ParameterElement.A2_TableFixtureCode[5])
      { S7_Templates := "SrcType := String" } NE_Contact(in1 := "AutoProcessData".A_Table_2[5].Code, in2 := '')
      wire#w6
      Move(in := 1, out1 => "AutoProcessData".A_Table_2[5].PartStatus)
   END_RUNG
   RUNG wire#w6
      Not()
      Move(in := 2, out1 => "AutoProcessData".A_Table_2[5].PartStatus)
   END_RUNG
   RUNG wire#w1
      { S7_Templates := "SrcType := String" } EQ_Contact(in1 := "AutoProcessData".A_Table_2[6].Code, in2 := "ST10_RecipeDB".ParameterElement.A2_TableFixtureCode[6])
      { S7_Templates := "SrcType := String" } NE_Contact(in1 := "AutoProcessData".A_Table_2[6].Code, in2 := '')
      wire#w7
      Move(in := 1, out1 => "AutoProcessData".A_Table_2[6].PartStatus)
   END_RUNG
   RUNG wire#w7
      Not()
      Move(in := 2, out1 => "AutoProcessData".A_Table_2[6].PartStatus)
   END_RUNG
   RUNG wire#w1
      { S7_Templates := "SrcType := String" } EQ_Contact(in1 := "AutoProcessData".A_Table_2[7].Code, in2 := "ST10_RecipeDB".ParameterElement.A2_TableFixtureCode[7])
      { S7_Templates := "SrcType := String" } NE_Contact(in1 := "AutoProcessData".A_Table_2[7].Code, in2 := '')
      wire#w8
      Move(in := 1, out1 => "AutoProcessData".A_Table_2[7].PartStatus)
   END_RUNG
   RUNG wire#w8
      Not()
      Move(in := 2, out1 => "AutoProcessData".A_Table_2[7].PartStatus)
   END_RUNG
   RUNG wire#w1
      { S7_Templates := "SrcType := String" } EQ_Contact(in1 := "AutoProcessData".A_Table_2[8].Code, in2 := "ST10_RecipeDB".ParameterElement.A2_TableFixtureCode[8])
      { S7_Templates := "SrcType := String" } NE_Contact(in1 := "AutoProcessData".A_Table_2[8].Code, in2 := '')
      wire#w9
      Move(in := 1, out1 => "AutoProcessData".A_Table_2[8].PartStatus)
   END_RUNG
   RUNG wire#w9
      Not()
      Move(in := 2, out1 => "AutoProcessData".A_Table_2[8].PartStatus)
   END_RUNG
   RUNG wire#w1
      { S7_Templates := "SrcType := Int" } EQ_Contact(in1 := "AutoProcessData".A_Table_2[1].PartStatus, in2 := 1)
      { S7_Templates := "SrcType := Int" } EQ_Contact(in1 := "AutoProcessData".A_Table_2[2].PartStatus, in2 := 1)
      { S7_Templates := "SrcType := Int" } EQ_Contact(in1 := "AutoProcessData".A_Table_2[3].PartStatus, in2 := 1)
      { S7_Templates := "SrcType := Int" } EQ_Contact(in1 := "AutoProcessData".A_Table_2[4].PartStatus, in2 := 1)
      { S7_Templates := "SrcType := Int" } EQ_Contact(in1 := "AutoProcessData".A_Table_2[5].PartStatus, in2 := 1)
      { S7_Templates := "SrcType := Int" } EQ_Contact(in1 := "AutoProcessData".A_Table_2[6].PartStatus, in2 := 1)
      { S7_Templates := "SrcType := Int" } EQ_Contact(in1 := "AutoProcessData".A_Table_2[7].PartStatus, in2 := 1)
      { S7_Templates := "SrcType := Int" } EQ_Contact(in1 := "AutoProcessData".A_Table_2[8].PartStatus, in2 := 1)
      wire#w10
      Coil( "AutoProcessData".GlobalData.Table2CodeOKFlag )
   END_RUNG
   RUNG wire#w1
      Contact( "ST10_GeneralData".FunctionDeSelect.Global.DeSelectPB_ScanFixture )
   END_RUNG wire#w10
   // the same network as SCL:
   #_w1 := "AlwaysTRUE" AND ("AutoProcessData".A_Table_2[1].Code = "ST10_RecipeDB".ParameterElement.A2_TableFixtureCode[1]) AND ("AutoProcessData".A_Table_2[1].Code <> '');
   IF #_w1 THEN "AutoProcessData".A_Table_2[1].PartStatus := 1; END_IF;
   IF NOT #_w1 THEN "AutoProcessData".A_Table_2[1].PartStatus := 2; END_IF;
   #_w2 := "AlwaysTRUE" AND ("AutoProcessData".A_Table_2[2].Code = "ST10_RecipeDB".ParameterElement.A2_TableFixtureCode[2]) AND ("AutoProcessData".A_Table_2[2].Code <> '');
   IF #_w2 THEN "AutoProcessData".A_Table_2[2].PartStatus := 1; END_IF;
   IF NOT #_w2 THEN "AutoProcessData".A_Table_2[2].PartStatus := 2; END_IF;
   #_w3 := "AlwaysTRUE" AND ("AutoProcessData".A_Table_2[3].Code = "ST10_RecipeDB".ParameterElement.A2_TableFixtureCode[3]) AND ("AutoProcessData".A_Table_2[3].Code <> '');
   IF #_w3 THEN "AutoProcessData".A_Table_2[3].PartStatus := 1; END_IF;
   IF NOT #_w3 THEN "AutoProcessData".A_Table_2[3].PartStatus := 2; END_IF;
   #_w4 := "AlwaysTRUE" AND ("AutoProcessData".A_Table_2[4].Code = "ST10_RecipeDB".ParameterElement.A2_TableFixtureCode[4]) AND ("AutoProcessData".A_Table_2[4].Code <> '');
   IF #_w4 THEN "AutoProcessData".A_Table_2[4].PartStatus := 1; END_IF;
   IF NOT #_w4 THEN "AutoProcessData".A_Table_2[4].PartStatus := 2; END_IF;
   #_w5 := "AlwaysTRUE" AND ("AutoProcessData".A_Table_2[5].Code = "ST10_RecipeDB".ParameterElement.A2_TableFixtureCode[5]) AND ("AutoProcessData".A_Table_2[5].Code <> '');
   IF #_w5 THEN "AutoProcessData".A_Table_2[5].PartStatus := 1; END_IF;
   IF NOT #_w5 THEN "AutoProcessData".A_Table_2[5].PartStatus := 2; END_IF;
   #_w6 := "AlwaysTRUE" AND ("AutoProcessData".A_Table_2[6].Code = "ST10_RecipeDB".ParameterElement.A2_TableFixtureCode[6]) AND ("AutoProcessData".A_Table_2[6].Code <> '');
   IF #_w6 THEN "AutoProcessData".A_Table_2[6].PartStatus := 1; END_IF;
   IF NOT #_w6 THEN "AutoProcessData".A_Table_2[6].PartStatus := 2; END_IF;
   #_w7 := "AlwaysTRUE" AND ("AutoProcessData".A_Table_2[7].Code = "ST10_RecipeDB".ParameterElement.A2_TableFixtureCode[7]) AND ("AutoProcessData".A_Table_2[7].Code <> '');
   IF #_w7 THEN "AutoProcessData".A_Table_2[7].PartStatus := 1; END_IF;
   IF NOT #_w7 THEN "AutoProcessData".A_Table_2[7].PartStatus := 2; END_IF;
   #_w8 := "AlwaysTRUE" AND ("AutoProcessData".A_Table_2[8].Code = "ST10_RecipeDB".ParameterElement.A2_TableFixtureCode[8]) AND ("AutoProcessData".A_Table_2[8].Code <> '');
   IF #_w8 THEN "AutoProcessData".A_Table_2[8].PartStatus := 1; END_IF;
   IF NOT #_w8 THEN "AutoProcessData".A_Table_2[8].PartStatus := 2; END_IF;
   "AutoProcessData".GlobalData.Table2CodeOKFlag := "AlwaysTRUE" AND ((("AutoProcessData".A_Table_2[1].PartStatus = 1) AND ("AutoProcessData".A_Table_2[2].PartStatus = 1) AND ("AutoProcessData".A_Table_2[3].PartStatus = 1) AND ("AutoProcessData".A_Table_2[4].PartStatus = 1) AND ("AutoProcessData".A_Table_2[5].PartStatus = 1) AND ("AutoProcessData".A_Table_2[6].PartStatus = 1) AND ("AutoProcessData".A_Table_2[7].PartStatus = 1) AND ("AutoProcessData".A_Table_2[8].PartStatus = 1)) OR "ST10_GeneralData".FunctionDeSelect.Global.DeSelectPB_ScanFixture);
END_REGION

REGION Network 18: Robot1Grip Code
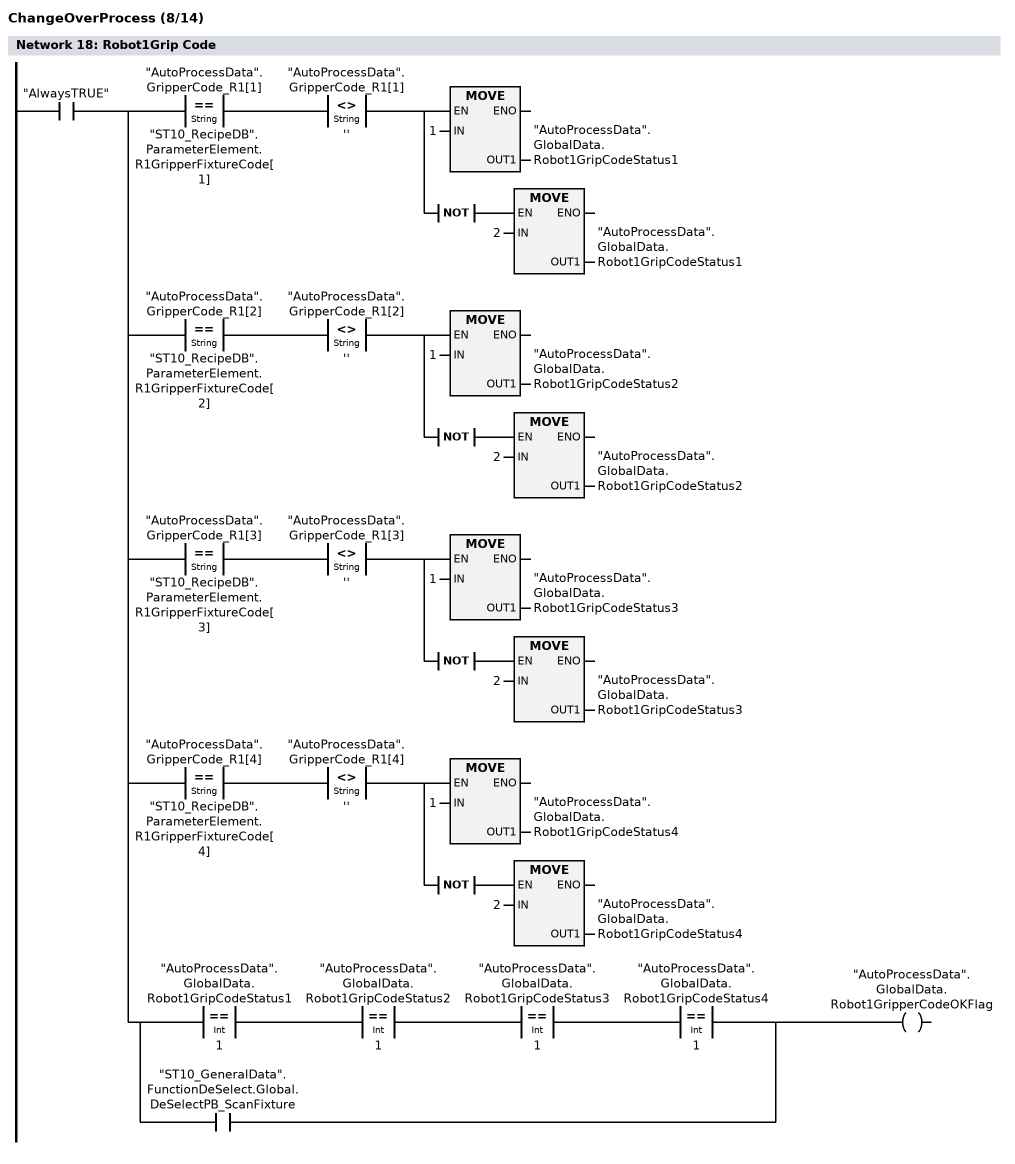
   RUNG wire#powerrail
      Contact( "AlwaysTRUE" )
      wire#w1
      { S7_Templates := "SrcType := String" } EQ_Contact(in1 := "AutoProcessData".GripperCode_R1[1], in2 := "ST10_RecipeDB".ParameterElement.R1GripperFixtureCode[1])
      { S7_Templates := "SrcType := String" } NE_Contact(in1 := "AutoProcessData".GripperCode_R1[1], in2 := '')
      wire#w2
      Move(in := 1, out1 => "AutoProcessData".GlobalData.Robot1GripCodeStatus1)
   END_RUNG
   RUNG wire#w2
      Not()
      Move(in := 2, out1 => "AutoProcessData".GlobalData.Robot1GripCodeStatus1)
   END_RUNG
   RUNG wire#w1
      { S7_Templates := "SrcType := String" } EQ_Contact(in1 := "AutoProcessData".GripperCode_R1[2], in2 := "ST10_RecipeDB".ParameterElement.R1GripperFixtureCode[2])
      { S7_Templates := "SrcType := String" } NE_Contact(in1 := "AutoProcessData".GripperCode_R1[2], in2 := '')
      wire#w3
      Move(in := 1, out1 => "AutoProcessData".GlobalData.Robot1GripCodeStatus2)
   END_RUNG
   RUNG wire#w3
      Not()
      Move(in := 2, out1 => "AutoProcessData".GlobalData.Robot1GripCodeStatus2)
   END_RUNG
   RUNG wire#w1
      { S7_Templates := "SrcType := String" } EQ_Contact(in1 := "AutoProcessData".GripperCode_R1[3], in2 := "ST10_RecipeDB".ParameterElement.R1GripperFixtureCode[3])
      { S7_Templates := "SrcType := String" } NE_Contact(in1 := "AutoProcessData".GripperCode_R1[3], in2 := '')
      wire#w4
      Move(in := 1, out1 => "AutoProcessData".GlobalData.Robot1GripCodeStatus3)
   END_RUNG
   RUNG wire#w4
      Not()
      Move(in := 2, out1 => "AutoProcessData".GlobalData.Robot1GripCodeStatus3)
   END_RUNG
   RUNG wire#w1
      { S7_Templates := "SrcType := String" } EQ_Contact(in1 := "AutoProcessData".GripperCode_R1[4], in2 := "ST10_RecipeDB".ParameterElement.R1GripperFixtureCode[4])
      { S7_Templates := "SrcType := String" } NE_Contact(in1 := "AutoProcessData".GripperCode_R1[4], in2 := '')
      wire#w5
      Move(in := 1, out1 => "AutoProcessData".GlobalData.Robot1GripCodeStatus4)
   END_RUNG
   RUNG wire#w5
      Not()
      Move(in := 2, out1 => "AutoProcessData".GlobalData.Robot1GripCodeStatus4)
   END_RUNG
   RUNG wire#w1
      { S7_Templates := "SrcType := Int" } EQ_Contact(in1 := "AutoProcessData".GlobalData.Robot1GripCodeStatus1, in2 := 1)
      { S7_Templates := "SrcType := Int" } EQ_Contact(in1 := "AutoProcessData".GlobalData.Robot1GripCodeStatus2, in2 := 1)
      { S7_Templates := "SrcType := Int" } EQ_Contact(in1 := "AutoProcessData".GlobalData.Robot1GripCodeStatus3, in2 := 1)
      { S7_Templates := "SrcType := Int" } EQ_Contact(in1 := "AutoProcessData".GlobalData.Robot1GripCodeStatus4, in2 := 1)
      wire#w6
      Coil( "AutoProcessData".GlobalData.Robot1GripperCodeOKFlag )
   END_RUNG
   RUNG wire#w1
      Contact( "ST10_GeneralData".FunctionDeSelect.Global.DeSelectPB_ScanFixture )
   END_RUNG wire#w6
   // the same network as SCL:
   #_w1 := "AlwaysTRUE" AND ("AutoProcessData".GripperCode_R1[1] = "ST10_RecipeDB".ParameterElement.R1GripperFixtureCode[1]) AND ("AutoProcessData".GripperCode_R1[1] <> '');
   IF #_w1 THEN "AutoProcessData".GlobalData.Robot1GripCodeStatus1 := 1; END_IF;
   IF NOT #_w1 THEN "AutoProcessData".GlobalData.Robot1GripCodeStatus1 := 2; END_IF;
   #_w2 := "AlwaysTRUE" AND ("AutoProcessData".GripperCode_R1[2] = "ST10_RecipeDB".ParameterElement.R1GripperFixtureCode[2]) AND ("AutoProcessData".GripperCode_R1[2] <> '');
   IF #_w2 THEN "AutoProcessData".GlobalData.Robot1GripCodeStatus2 := 1; END_IF;
   IF NOT #_w2 THEN "AutoProcessData".GlobalData.Robot1GripCodeStatus2 := 2; END_IF;
   #_w3 := "AlwaysTRUE" AND ("AutoProcessData".GripperCode_R1[3] = "ST10_RecipeDB".ParameterElement.R1GripperFixtureCode[3]) AND ("AutoProcessData".GripperCode_R1[3] <> '');
   IF #_w3 THEN "AutoProcessData".GlobalData.Robot1GripCodeStatus3 := 1; END_IF;
   IF NOT #_w3 THEN "AutoProcessData".GlobalData.Robot1GripCodeStatus3 := 2; END_IF;
   #_w4 := "AlwaysTRUE" AND ("AutoProcessData".GripperCode_R1[4] = "ST10_RecipeDB".ParameterElement.R1GripperFixtureCode[4]) AND ("AutoProcessData".GripperCode_R1[4] <> '');
   IF #_w4 THEN "AutoProcessData".GlobalData.Robot1GripCodeStatus4 := 1; END_IF;
   IF NOT #_w4 THEN "AutoProcessData".GlobalData.Robot1GripCodeStatus4 := 2; END_IF;
   "AutoProcessData".GlobalData.Robot1GripperCodeOKFlag := "AlwaysTRUE" AND ((("AutoProcessData".GlobalData.Robot1GripCodeStatus1 = 1) AND ("AutoProcessData".GlobalData.Robot1GripCodeStatus2 = 1) AND ("AutoProcessData".GlobalData.Robot1GripCodeStatus3 = 1) AND ("AutoProcessData".GlobalData.Robot1GripCodeStatus4 = 1)) OR "ST10_GeneralData".FunctionDeSelect.Global.DeSelectPB_ScanFixture);
END_REGION

REGION Network 19: Robot2Grip Code
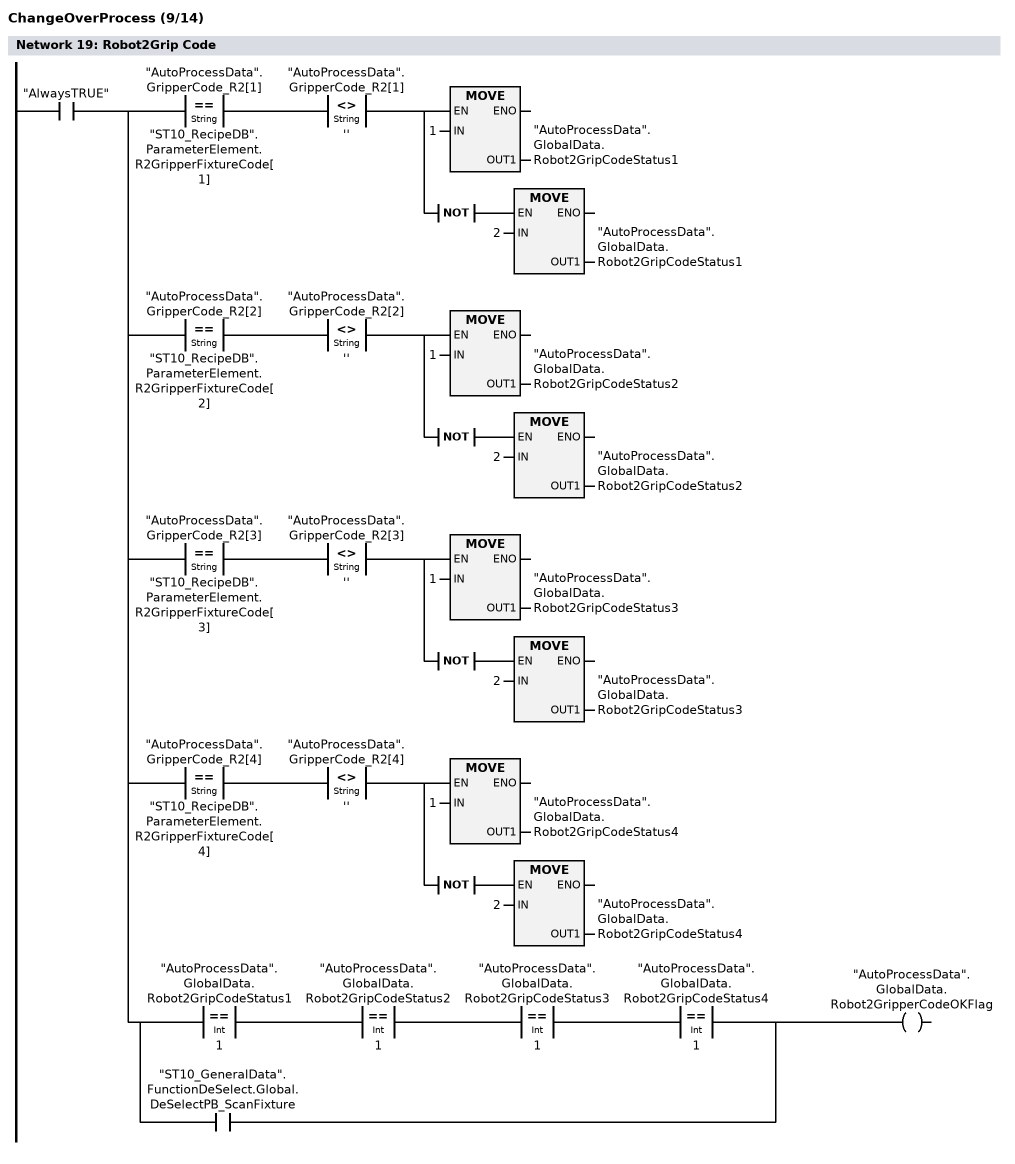
   RUNG wire#powerrail
      Contact( "AlwaysTRUE" )
      wire#w1
      { S7_Templates := "SrcType := String" } EQ_Contact(in1 := "AutoProcessData".GripperCode_R2[1], in2 := "ST10_RecipeDB".ParameterElement.R2GripperFixtureCode[1])
      { S7_Templates := "SrcType := String" } NE_Contact(in1 := "AutoProcessData".GripperCode_R2[1], in2 := '')
      wire#w2
      Move(in := 1, out1 => "AutoProcessData".GlobalData.Robot2GripCodeStatus1)
   END_RUNG
   RUNG wire#w2
      Not()
      Move(in := 2, out1 => "AutoProcessData".GlobalData.Robot2GripCodeStatus1)
   END_RUNG
   RUNG wire#w1
      { S7_Templates := "SrcType := String" } EQ_Contact(in1 := "AutoProcessData".GripperCode_R2[2], in2 := "ST10_RecipeDB".ParameterElement.R2GripperFixtureCode[2])
      { S7_Templates := "SrcType := String" } NE_Contact(in1 := "AutoProcessData".GripperCode_R2[2], in2 := '')
      wire#w3
      Move(in := 1, out1 => "AutoProcessData".GlobalData.Robot2GripCodeStatus2)
   END_RUNG
   RUNG wire#w3
      Not()
      Move(in := 2, out1 => "AutoProcessData".GlobalData.Robot2GripCodeStatus2)
   END_RUNG
   RUNG wire#w1
      { S7_Templates := "SrcType := String" } EQ_Contact(in1 := "AutoProcessData".GripperCode_R2[3], in2 := "ST10_RecipeDB".ParameterElement.R2GripperFixtureCode[3])
      { S7_Templates := "SrcType := String" } NE_Contact(in1 := "AutoProcessData".GripperCode_R2[3], in2 := '')
      wire#w4
      Move(in := 1, out1 => "AutoProcessData".GlobalData.Robot2GripCodeStatus3)
   END_RUNG
   RUNG wire#w4
      Not()
      Move(in := 2, out1 => "AutoProcessData".GlobalData.Robot2GripCodeStatus3)
   END_RUNG
   RUNG wire#w1
      { S7_Templates := "SrcType := String" } EQ_Contact(in1 := "AutoProcessData".GripperCode_R2[4], in2 := "ST10_RecipeDB".ParameterElement.R2GripperFixtureCode[4])
      { S7_Templates := "SrcType := String" } NE_Contact(in1 := "AutoProcessData".GripperCode_R2[4], in2 := '')
      wire#w5
      Move(in := 1, out1 => "AutoProcessData".GlobalData.Robot2GripCodeStatus4)
   END_RUNG
   RUNG wire#w5
      Not()
      Move(in := 2, out1 => "AutoProcessData".GlobalData.Robot2GripCodeStatus4)
   END_RUNG
   RUNG wire#w1
      { S7_Templates := "SrcType := Int" } EQ_Contact(in1 := "AutoProcessData".GlobalData.Robot2GripCodeStatus1, in2 := 1)
      { S7_Templates := "SrcType := Int" } EQ_Contact(in1 := "AutoProcessData".GlobalData.Robot2GripCodeStatus2, in2 := 1)
      { S7_Templates := "SrcType := Int" } EQ_Contact(in1 := "AutoProcessData".GlobalData.Robot2GripCodeStatus3, in2 := 1)
      { S7_Templates := "SrcType := Int" } EQ_Contact(in1 := "AutoProcessData".GlobalData.Robot2GripCodeStatus4, in2 := 1)
      wire#w6
      Coil( "AutoProcessData".GlobalData.Robot2GripperCodeOKFlag )
   END_RUNG
   RUNG wire#w1
      Contact( "ST10_GeneralData".FunctionDeSelect.Global.DeSelectPB_ScanFixture )
   END_RUNG wire#w6
   // the same network as SCL:
   #_w1 := "AlwaysTRUE" AND ("AutoProcessData".GripperCode_R2[1] = "ST10_RecipeDB".ParameterElement.R2GripperFixtureCode[1]) AND ("AutoProcessData".GripperCode_R2[1] <> '');
   IF #_w1 THEN "AutoProcessData".GlobalData.Robot2GripCodeStatus1 := 1; END_IF;
   IF NOT #_w1 THEN "AutoProcessData".GlobalData.Robot2GripCodeStatus1 := 2; END_IF;
   #_w2 := "AlwaysTRUE" AND ("AutoProcessData".GripperCode_R2[2] = "ST10_RecipeDB".ParameterElement.R2GripperFixtureCode[2]) AND ("AutoProcessData".GripperCode_R2[2] <> '');
   IF #_w2 THEN "AutoProcessData".GlobalData.Robot2GripCodeStatus2 := 1; END_IF;
   IF NOT #_w2 THEN "AutoProcessData".GlobalData.Robot2GripCodeStatus2 := 2; END_IF;
   #_w3 := "AlwaysTRUE" AND ("AutoProcessData".GripperCode_R2[3] = "ST10_RecipeDB".ParameterElement.R2GripperFixtureCode[3]) AND ("AutoProcessData".GripperCode_R2[3] <> '');
   IF #_w3 THEN "AutoProcessData".GlobalData.Robot2GripCodeStatus3 := 1; END_IF;
   IF NOT #_w3 THEN "AutoProcessData".GlobalData.Robot2GripCodeStatus3 := 2; END_IF;
   #_w4 := "AlwaysTRUE" AND ("AutoProcessData".GripperCode_R2[4] = "ST10_RecipeDB".ParameterElement.R2GripperFixtureCode[4]) AND ("AutoProcessData".GripperCode_R2[4] <> '');
   IF #_w4 THEN "AutoProcessData".GlobalData.Robot2GripCodeStatus4 := 1; END_IF;
   IF NOT #_w4 THEN "AutoProcessData".GlobalData.Robot2GripCodeStatus4 := 2; END_IF;
   "AutoProcessData".GlobalData.Robot2GripperCodeOKFlag := "AlwaysTRUE" AND ((("AutoProcessData".GlobalData.Robot2GripCodeStatus1 = 1) AND ("AutoProcessData".GlobalData.Robot2GripCodeStatus2 = 1) AND ("AutoProcessData".GlobalData.Robot2GripCodeStatus3 = 1) AND ("AutoProcessData".GlobalData.Robot2GripCodeStatus4 = 1)) OR "ST10_GeneralData".FunctionDeSelect.Global.DeSelectPB_ScanFixture);
END_REGION

REGION Network 20: Robot3Grip Code
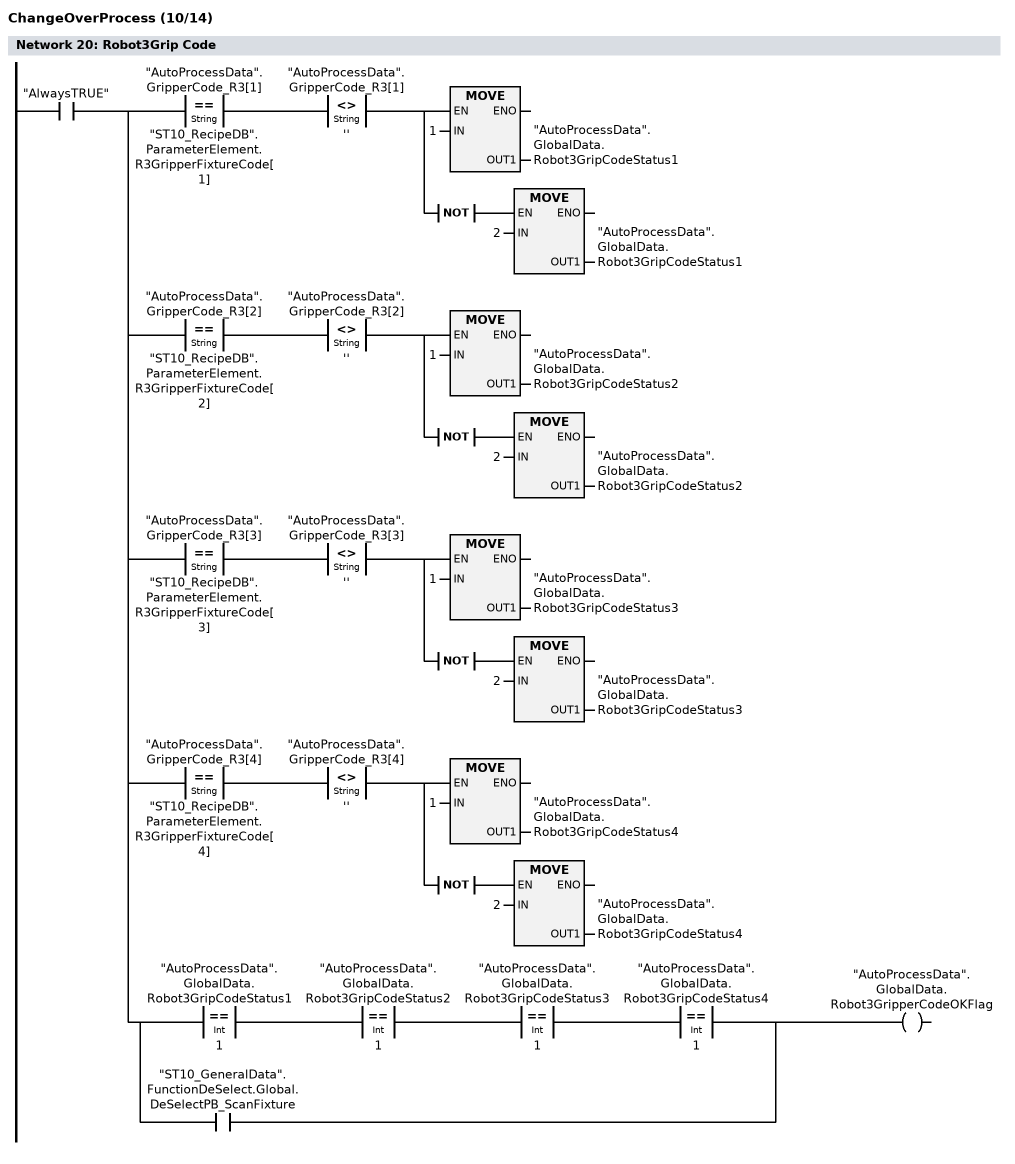
   RUNG wire#powerrail
      Contact( "AlwaysTRUE" )
      wire#w1
      { S7_Templates := "SrcType := String" } EQ_Contact(in1 := "AutoProcessData".GripperCode_R3[1], in2 := "ST10_RecipeDB".ParameterElement.R3GripperFixtureCode[1])
      { S7_Templates := "SrcType := String" } NE_Contact(in1 := "AutoProcessData".GripperCode_R3[1], in2 := '')
      wire#w2
      Move(in := 1, out1 => "AutoProcessData".GlobalData.Robot3GripCodeStatus1)
   END_RUNG
   RUNG wire#w2
      Not()
      Move(in := 2, out1 => "AutoProcessData".GlobalData.Robot3GripCodeStatus1)
   END_RUNG
   RUNG wire#w1
      { S7_Templates := "SrcType := String" } EQ_Contact(in1 := "AutoProcessData".GripperCode_R3[2], in2 := "ST10_RecipeDB".ParameterElement.R3GripperFixtureCode[2])
      { S7_Templates := "SrcType := String" } NE_Contact(in1 := "AutoProcessData".GripperCode_R3[2], in2 := '')
      wire#w3
      Move(in := 1, out1 => "AutoProcessData".GlobalData.Robot3GripCodeStatus2)
   END_RUNG
   RUNG wire#w3
      Not()
      Move(in := 2, out1 => "AutoProcessData".GlobalData.Robot3GripCodeStatus2)
   END_RUNG
   RUNG wire#w1
      { S7_Templates := "SrcType := String" } EQ_Contact(in1 := "AutoProcessData".GripperCode_R3[3], in2 := "ST10_RecipeDB".ParameterElement.R3GripperFixtureCode[3])
      { S7_Templates := "SrcType := String" } NE_Contact(in1 := "AutoProcessData".GripperCode_R3[3], in2 := '')
      wire#w4
      Move(in := 1, out1 => "AutoProcessData".GlobalData.Robot3GripCodeStatus3)
   END_RUNG
   RUNG wire#w4
      Not()
      Move(in := 2, out1 => "AutoProcessData".GlobalData.Robot3GripCodeStatus3)
   END_RUNG
   RUNG wire#w1
      { S7_Templates := "SrcType := String" } EQ_Contact(in1 := "AutoProcessData".GripperCode_R3[4], in2 := "ST10_RecipeDB".ParameterElement.R3GripperFixtureCode[4])
      { S7_Templates := "SrcType := String" } NE_Contact(in1 := "AutoProcessData".GripperCode_R3[4], in2 := '')
      wire#w5
      Move(in := 1, out1 => "AutoProcessData".GlobalData.Robot3GripCodeStatus4)
   END_RUNG
   RUNG wire#w5
      Not()
      Move(in := 2, out1 => "AutoProcessData".GlobalData.Robot3GripCodeStatus4)
   END_RUNG
   RUNG wire#w1
      { S7_Templates := "SrcType := Int" } EQ_Contact(in1 := "AutoProcessData".GlobalData.Robot3GripCodeStatus1, in2 := 1)
      { S7_Templates := "SrcType := Int" } EQ_Contact(in1 := "AutoProcessData".GlobalData.Robot3GripCodeStatus2, in2 := 1)
      { S7_Templates := "SrcType := Int" } EQ_Contact(in1 := "AutoProcessData".GlobalData.Robot3GripCodeStatus3, in2 := 1)
      { S7_Templates := "SrcType := Int" } EQ_Contact(in1 := "AutoProcessData".GlobalData.Robot3GripCodeStatus4, in2 := 1)
      wire#w6
      Coil( "AutoProcessData".GlobalData.Robot3GripperCodeOKFlag )
   END_RUNG
   RUNG wire#w1
      Contact( "ST10_GeneralData".FunctionDeSelect.Global.DeSelectPB_ScanFixture )
   END_RUNG wire#w6
   // the same network as SCL:
   #_w1 := "AlwaysTRUE" AND ("AutoProcessData".GripperCode_R3[1] = "ST10_RecipeDB".ParameterElement.R3GripperFixtureCode[1]) AND ("AutoProcessData".GripperCode_R3[1] <> '');
   IF #_w1 THEN "AutoProcessData".GlobalData.Robot3GripCodeStatus1 := 1; END_IF;
   IF NOT #_w1 THEN "AutoProcessData".GlobalData.Robot3GripCodeStatus1 := 2; END_IF;
   #_w2 := "AlwaysTRUE" AND ("AutoProcessData".GripperCode_R3[2] = "ST10_RecipeDB".ParameterElement.R3GripperFixtureCode[2]) AND ("AutoProcessData".GripperCode_R3[2] <> '');
   IF #_w2 THEN "AutoProcessData".GlobalData.Robot3GripCodeStatus2 := 1; END_IF;
   IF NOT #_w2 THEN "AutoProcessData".GlobalData.Robot3GripCodeStatus2 := 2; END_IF;
   #_w3 := "AlwaysTRUE" AND ("AutoProcessData".GripperCode_R3[3] = "ST10_RecipeDB".ParameterElement.R3GripperFixtureCode[3]) AND ("AutoProcessData".GripperCode_R3[3] <> '');
   IF #_w3 THEN "AutoProcessData".GlobalData.Robot3GripCodeStatus3 := 1; END_IF;
   IF NOT #_w3 THEN "AutoProcessData".GlobalData.Robot3GripCodeStatus3 := 2; END_IF;
   #_w4 := "AlwaysTRUE" AND ("AutoProcessData".GripperCode_R3[4] = "ST10_RecipeDB".ParameterElement.R3GripperFixtureCode[4]) AND ("AutoProcessData".GripperCode_R3[4] <> '');
   IF #_w4 THEN "AutoProcessData".GlobalData.Robot3GripCodeStatus4 := 1; END_IF;
   IF NOT #_w4 THEN "AutoProcessData".GlobalData.Robot3GripCodeStatus4 := 2; END_IF;
   "AutoProcessData".GlobalData.Robot3GripperCodeOKFlag := "AlwaysTRUE" AND ((("AutoProcessData".GlobalData.Robot3GripCodeStatus1 = 1) AND ("AutoProcessData".GlobalData.Robot3GripCodeStatus2 = 1) AND ("AutoProcessData".GlobalData.Robot3GripCodeStatus3 = 1) AND ("AutoProcessData".GlobalData.Robot3GripCodeStatus4 = 1)) OR "ST10_GeneralData".FunctionDeSelect.Global.DeSelectPB_ScanFixture);
END_REGION

REGION Network 21: A1 Fixture Code
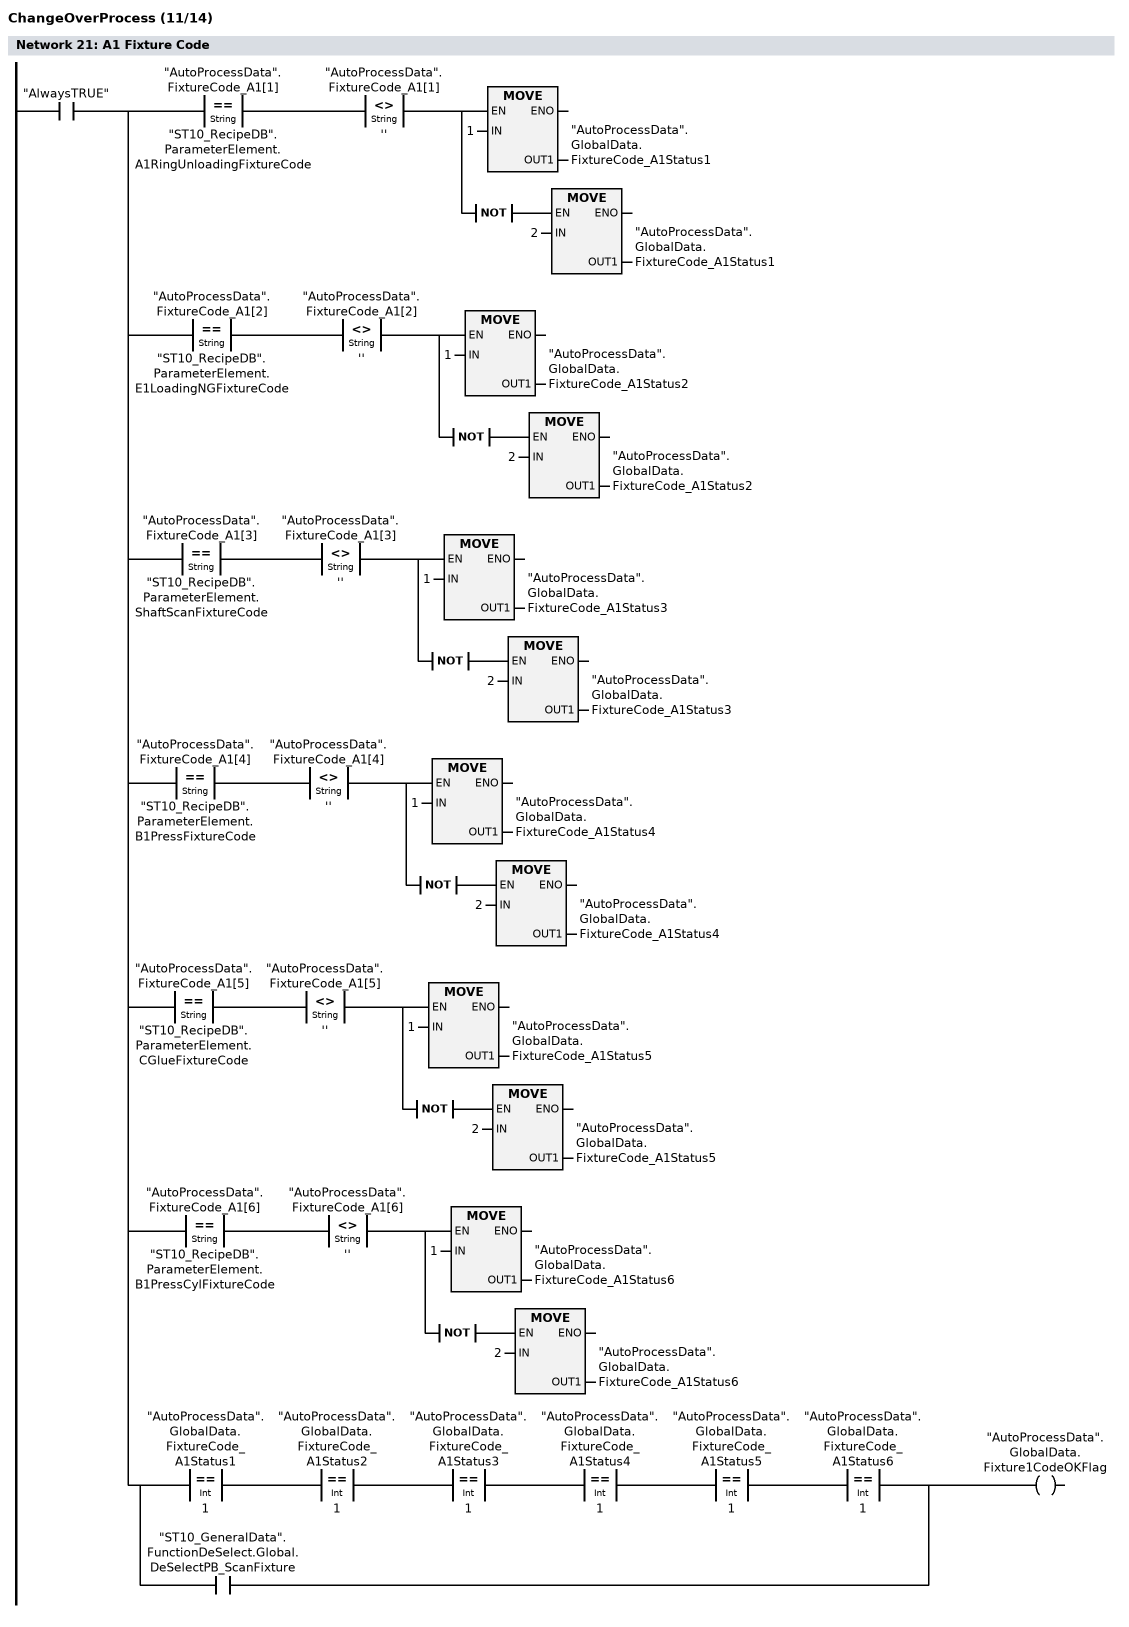
   RUNG wire#powerrail
      Contact( "AlwaysTRUE" )
      wire#w1
      { S7_Templates := "SrcType := String" } EQ_Contact(in1 := "AutoProcessData".FixtureCode_A1[1], in2 := "ST10_RecipeDB".ParameterElement.A1RingUnloadingFixtureCode)
      { S7_Templates := "SrcType := String" } NE_Contact(in1 := "AutoProcessData".FixtureCode_A1[1], in2 := '')
      wire#w2
      Move(in := 1, out1 => "AutoProcessData".GlobalData.FixtureCode_A1Status1)
   END_RUNG
   RUNG wire#w2
      Not()
      Move(in := 2, out1 => "AutoProcessData".GlobalData.FixtureCode_A1Status1)
   END_RUNG
   RUNG wire#w1
      { S7_Templates := "SrcType := String" } EQ_Contact(in1 := "AutoProcessData".FixtureCode_A1[2], in2 := "ST10_RecipeDB".ParameterElement.E1LoadingNGFixtureCode)
      { S7_Templates := "SrcType := String" } NE_Contact(in1 := "AutoProcessData".FixtureCode_A1[2], in2 := '')
      wire#w3
      Move(in := 1, out1 => "AutoProcessData".GlobalData.FixtureCode_A1Status2)
   END_RUNG
   RUNG wire#w3
      Not()
      Move(in := 2, out1 => "AutoProcessData".GlobalData.FixtureCode_A1Status2)
   END_RUNG
   RUNG wire#w1
      { S7_Templates := "SrcType := String" } EQ_Contact(in1 := "AutoProcessData".FixtureCode_A1[3], in2 := "ST10_RecipeDB".ParameterElement.ShaftScanFixtureCode)
      { S7_Templates := "SrcType := String" } NE_Contact(in1 := "AutoProcessData".FixtureCode_A1[3], in2 := '')
      wire#w4
      Move(in := 1, out1 => "AutoProcessData".GlobalData.FixtureCode_A1Status3)
   END_RUNG
   RUNG wire#w4
      Not()
      Move(in := 2, out1 => "AutoProcessData".GlobalData.FixtureCode_A1Status3)
   END_RUNG
   RUNG wire#w1
      { S7_Templates := "SrcType := String" } EQ_Contact(in1 := "AutoProcessData".FixtureCode_A1[4], in2 := "ST10_RecipeDB".ParameterElement.B1PressFixtureCode)
      { S7_Templates := "SrcType := String" } NE_Contact(in1 := "AutoProcessData".FixtureCode_A1[4], in2 := '')
      wire#w5
      Move(in := 1, out1 => "AutoProcessData".GlobalData.FixtureCode_A1Status4)
   END_RUNG
   RUNG wire#w5
      Not()
      Move(in := 2, out1 => "AutoProcessData".GlobalData.FixtureCode_A1Status4)
   END_RUNG
   RUNG wire#w1
      { S7_Templates := "SrcType := String" } EQ_Contact(in1 := "AutoProcessData".FixtureCode_A1[5], in2 := "ST10_RecipeDB".ParameterElement.CGlueFixtureCode)
      { S7_Templates := "SrcType := String" } NE_Contact(in1 := "AutoProcessData".FixtureCode_A1[5], in2 := '')
      wire#w6
      Move(in := 1, out1 => "AutoProcessData".GlobalData.FixtureCode_A1Status5)
   END_RUNG
   RUNG wire#w6
      Not()
      Move(in := 2, out1 => "AutoProcessData".GlobalData.FixtureCode_A1Status5)
   END_RUNG
   RUNG wire#w1
      { S7_Templates := "SrcType := String" } EQ_Contact(in1 := "AutoProcessData".FixtureCode_A1[6], in2 := "ST10_RecipeDB".ParameterElement.B1PressCylFixtureCode)
      { S7_Templates := "SrcType := String" } NE_Contact(in1 := "AutoProcessData".FixtureCode_A1[6], in2 := '')
      wire#w7
      Move(in := 1, out1 => "AutoProcessData".GlobalData.FixtureCode_A1Status6)
   END_RUNG
   RUNG wire#w7
      Not()
      Move(in := 2, out1 => "AutoProcessData".GlobalData.FixtureCode_A1Status6)
   END_RUNG
   RUNG wire#w1
      { S7_Templates := "SrcType := Int" } EQ_Contact(in1 := "AutoProcessData".GlobalData.FixtureCode_A1Status1, in2 := 1)
      { S7_Templates := "SrcType := Int" } EQ_Contact(in1 := "AutoProcessData".GlobalData.FixtureCode_A1Status2, in2 := 1)
      { S7_Templates := "SrcType := Int" } EQ_Contact(in1 := "AutoProcessData".GlobalData.FixtureCode_A1Status3, in2 := 1)
      { S7_Templates := "SrcType := Int" } EQ_Contact(in1 := "AutoProcessData".GlobalData.FixtureCode_A1Status4, in2 := 1)
      { S7_Templates := "SrcType := Int" } EQ_Contact(in1 := "AutoProcessData".GlobalData.FixtureCode_A1Status5, in2 := 1)
      { S7_Templates := "SrcType := Int" } EQ_Contact(in1 := "AutoProcessData".GlobalData.FixtureCode_A1Status6, in2 := 1)
      wire#w8
      Coil( "AutoProcessData".GlobalData.Fixture1CodeOKFlag )
   END_RUNG
   RUNG wire#w1
      Contact( "ST10_GeneralData".FunctionDeSelect.Global.DeSelectPB_ScanFixture )
   END_RUNG wire#w8
   // the same network as SCL:
   #_w1 := "AlwaysTRUE" AND ("AutoProcessData".FixtureCode_A1[1] = "ST10_RecipeDB".ParameterElement.A1RingUnloadingFixtureCode) AND ("AutoProcessData".FixtureCode_A1[1] <> '');
   IF #_w1 THEN "AutoProcessData".GlobalData.FixtureCode_A1Status1 := 1; END_IF;
   IF NOT #_w1 THEN "AutoProcessData".GlobalData.FixtureCode_A1Status1 := 2; END_IF;
   #_w2 := "AlwaysTRUE" AND ("AutoProcessData".FixtureCode_A1[2] = "ST10_RecipeDB".ParameterElement.E1LoadingNGFixtureCode) AND ("AutoProcessData".FixtureCode_A1[2] <> '');
   IF #_w2 THEN "AutoProcessData".GlobalData.FixtureCode_A1Status2 := 1; END_IF;
   IF NOT #_w2 THEN "AutoProcessData".GlobalData.FixtureCode_A1Status2 := 2; END_IF;
   #_w3 := "AlwaysTRUE" AND ("AutoProcessData".FixtureCode_A1[3] = "ST10_RecipeDB".ParameterElement.ShaftScanFixtureCode) AND ("AutoProcessData".FixtureCode_A1[3] <> '');
   IF #_w3 THEN "AutoProcessData".GlobalData.FixtureCode_A1Status3 := 1; END_IF;
   IF NOT #_w3 THEN "AutoProcessData".GlobalData.FixtureCode_A1Status3 := 2; END_IF;
   #_w4 := "AlwaysTRUE" AND ("AutoProcessData".FixtureCode_A1[4] = "ST10_RecipeDB".ParameterElement.B1PressFixtureCode) AND ("AutoProcessData".FixtureCode_A1[4] <> '');
   IF #_w4 THEN "AutoProcessData".GlobalData.FixtureCode_A1Status4 := 1; END_IF;
   IF NOT #_w4 THEN "AutoProcessData".GlobalData.FixtureCode_A1Status4 := 2; END_IF;
   #_w5 := "AlwaysTRUE" AND ("AutoProcessData".FixtureCode_A1[5] = "ST10_RecipeDB".ParameterElement.CGlueFixtureCode) AND ("AutoProcessData".FixtureCode_A1[5] <> '');
   IF #_w5 THEN "AutoProcessData".GlobalData.FixtureCode_A1Status5 := 1; END_IF;
   IF NOT #_w5 THEN "AutoProcessData".GlobalData.FixtureCode_A1Status5 := 2; END_IF;
   #_w6 := "AlwaysTRUE" AND ("AutoProcessData".FixtureCode_A1[6] = "ST10_RecipeDB".ParameterElement.B1PressCylFixtureCode) AND ("AutoProcessData".FixtureCode_A1[6] <> '');
   IF #_w6 THEN "AutoProcessData".GlobalData.FixtureCode_A1Status6 := 1; END_IF;
   IF NOT #_w6 THEN "AutoProcessData".GlobalData.FixtureCode_A1Status6 := 2; END_IF;
   "AutoProcessData".GlobalData.Fixture1CodeOKFlag := "AlwaysTRUE" AND ((("AutoProcessData".GlobalData.FixtureCode_A1Status1 = 1) AND ("AutoProcessData".GlobalData.FixtureCode_A1Status2 = 1) AND ("AutoProcessData".GlobalData.FixtureCode_A1Status3 = 1) AND ("AutoProcessData".GlobalData.FixtureCode_A1Status4 = 1) AND ("AutoProcessData".GlobalData.FixtureCode_A1Status5 = 1) AND ("AutoProcessData".GlobalData.FixtureCode_A1Status6 = 1)) OR "ST10_GeneralData".FunctionDeSelect.Global.DeSelectPB_ScanFixture);
END_REGION

REGION Network 22: A2 Fixture Code
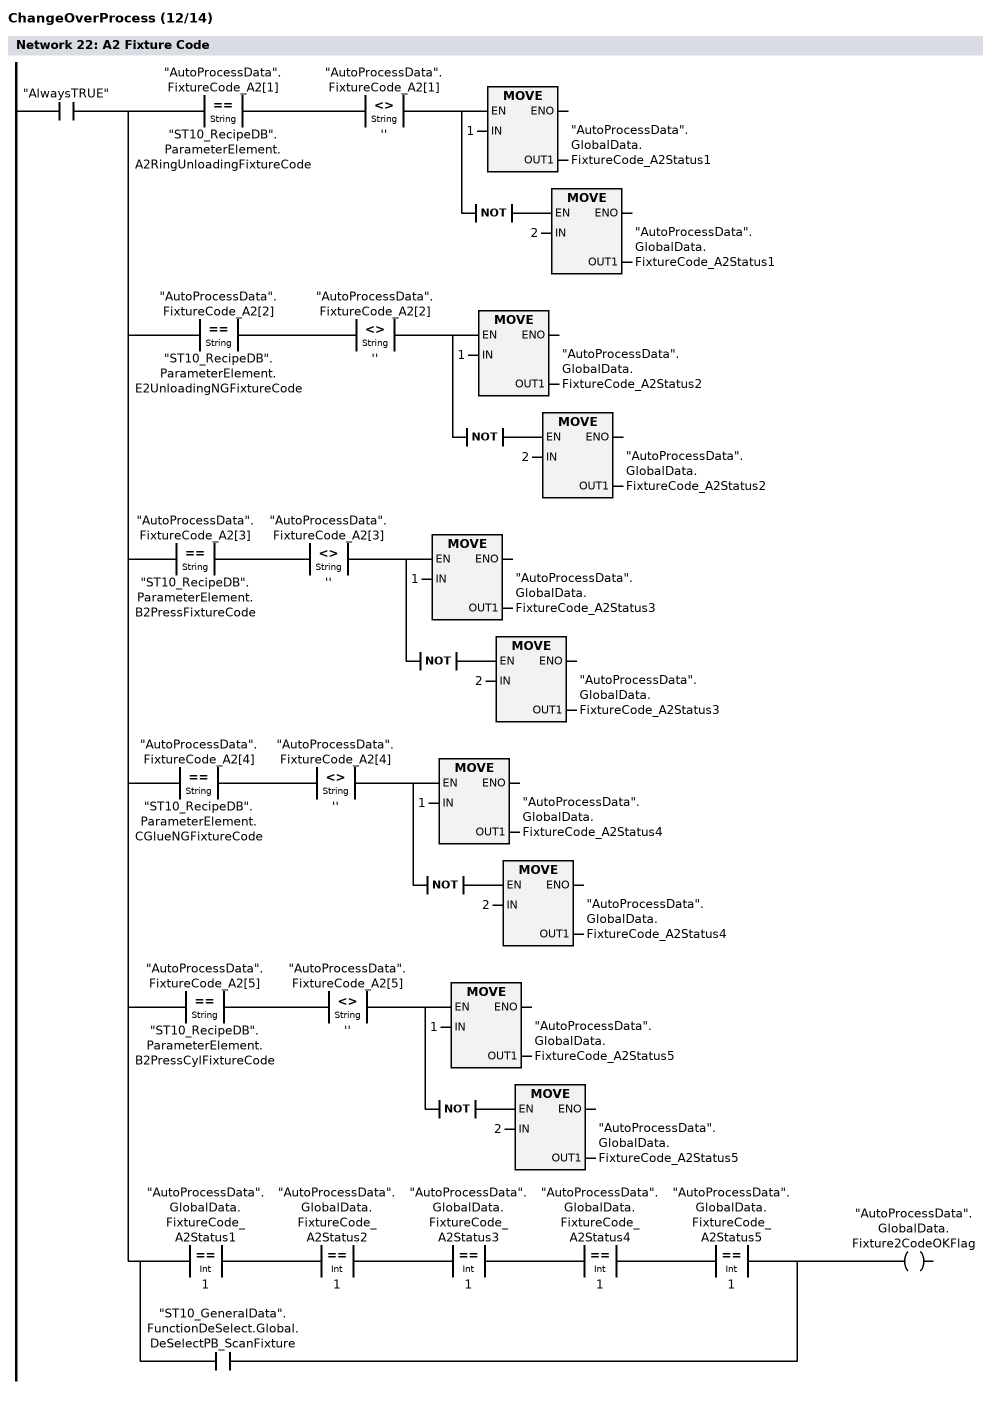
   RUNG wire#powerrail
      Contact( "AlwaysTRUE" )
      wire#w1
      { S7_Templates := "SrcType := String" } EQ_Contact(in1 := "AutoProcessData".FixtureCode_A2[1], in2 := "ST10_RecipeDB".ParameterElement.A2RingUnloadingFixtureCode)
      { S7_Templates := "SrcType := String" } NE_Contact(in1 := "AutoProcessData".FixtureCode_A2[1], in2 := '')
      wire#w2
      Move(in := 1, out1 => "AutoProcessData".GlobalData.FixtureCode_A2Status1)
   END_RUNG
   RUNG wire#w2
      Not()
      Move(in := 2, out1 => "AutoProcessData".GlobalData.FixtureCode_A2Status1)
   END_RUNG
   RUNG wire#w1
      { S7_Templates := "SrcType := String" } EQ_Contact(in1 := "AutoProcessData".FixtureCode_A2[2], in2 := "ST10_RecipeDB".ParameterElement.E2UnloadingNGFixtureCode)
      { S7_Templates := "SrcType := String" } NE_Contact(in1 := "AutoProcessData".FixtureCode_A2[2], in2 := '')
      wire#w3
      Move(in := 1, out1 => "AutoProcessData".GlobalData.FixtureCode_A2Status2)
   END_RUNG
   RUNG wire#w3
      Not()
      Move(in := 2, out1 => "AutoProcessData".GlobalData.FixtureCode_A2Status2)
   END_RUNG
   RUNG wire#w1
      { S7_Templates := "SrcType := String" } EQ_Contact(in1 := "AutoProcessData".FixtureCode_A2[3], in2 := "ST10_RecipeDB".ParameterElement.B2PressFixtureCode)
      { S7_Templates := "SrcType := String" } NE_Contact(in1 := "AutoProcessData".FixtureCode_A2[3], in2 := '')
      wire#w4
      Move(in := 1, out1 => "AutoProcessData".GlobalData.FixtureCode_A2Status3)
   END_RUNG
   RUNG wire#w4
      Not()
      Move(in := 2, out1 => "AutoProcessData".GlobalData.FixtureCode_A2Status3)
   END_RUNG
   RUNG wire#w1
      { S7_Templates := "SrcType := String" } EQ_Contact(in1 := "AutoProcessData".FixtureCode_A2[4], in2 := "ST10_RecipeDB".ParameterElement.CGlueNGFixtureCode)
      { S7_Templates := "SrcType := String" } NE_Contact(in1 := "AutoProcessData".FixtureCode_A2[4], in2 := '')
      wire#w5
      Move(in := 1, out1 => "AutoProcessData".GlobalData.FixtureCode_A2Status4)
   END_RUNG
   RUNG wire#w5
      Not()
      Move(in := 2, out1 => "AutoProcessData".GlobalData.FixtureCode_A2Status4)
   END_RUNG
   RUNG wire#w1
      { S7_Templates := "SrcType := String" } EQ_Contact(in1 := "AutoProcessData".FixtureCode_A2[5], in2 := "ST10_RecipeDB".ParameterElement.B2PressCylFixtureCode)
      { S7_Templates := "SrcType := String" } NE_Contact(in1 := "AutoProcessData".FixtureCode_A2[5], in2 := '')
      wire#w6
      Move(in := 1, out1 => "AutoProcessData".GlobalData.FixtureCode_A2Status5)
   END_RUNG
   RUNG wire#w6
      Not()
      Move(in := 2, out1 => "AutoProcessData".GlobalData.FixtureCode_A2Status5)
   END_RUNG
   RUNG wire#w1
      { S7_Templates := "SrcType := Int" } EQ_Contact(in1 := "AutoProcessData".GlobalData.FixtureCode_A2Status1, in2 := 1)
      { S7_Templates := "SrcType := Int" } EQ_Contact(in1 := "AutoProcessData".GlobalData.FixtureCode_A2Status2, in2 := 1)
      { S7_Templates := "SrcType := Int" } EQ_Contact(in1 := "AutoProcessData".GlobalData.FixtureCode_A2Status3, in2 := 1)
      { S7_Templates := "SrcType := Int" } EQ_Contact(in1 := "AutoProcessData".GlobalData.FixtureCode_A2Status4, in2 := 1)
      { S7_Templates := "SrcType := Int" } EQ_Contact(in1 := "AutoProcessData".GlobalData.FixtureCode_A2Status5, in2 := 1)
      wire#w7
      Coil( "AutoProcessData".GlobalData.Fixture2CodeOKFlag )
   END_RUNG
   RUNG wire#w1
      Contact( "ST10_GeneralData".FunctionDeSelect.Global.DeSelectPB_ScanFixture )
   END_RUNG wire#w7
   // the same network as SCL:
   #_w1 := "AlwaysTRUE" AND ("AutoProcessData".FixtureCode_A2[1] = "ST10_RecipeDB".ParameterElement.A2RingUnloadingFixtureCode) AND ("AutoProcessData".FixtureCode_A2[1] <> '');
   IF #_w1 THEN "AutoProcessData".GlobalData.FixtureCode_A2Status1 := 1; END_IF;
   IF NOT #_w1 THEN "AutoProcessData".GlobalData.FixtureCode_A2Status1 := 2; END_IF;
   #_w2 := "AlwaysTRUE" AND ("AutoProcessData".FixtureCode_A2[2] = "ST10_RecipeDB".ParameterElement.E2UnloadingNGFixtureCode) AND ("AutoProcessData".FixtureCode_A2[2] <> '');
   IF #_w2 THEN "AutoProcessData".GlobalData.FixtureCode_A2Status2 := 1; END_IF;
   IF NOT #_w2 THEN "AutoProcessData".GlobalData.FixtureCode_A2Status2 := 2; END_IF;
   #_w3 := "AlwaysTRUE" AND ("AutoProcessData".FixtureCode_A2[3] = "ST10_RecipeDB".ParameterElement.B2PressFixtureCode) AND ("AutoProcessData".FixtureCode_A2[3] <> '');
   IF #_w3 THEN "AutoProcessData".GlobalData.FixtureCode_A2Status3 := 1; END_IF;
   IF NOT #_w3 THEN "AutoProcessData".GlobalData.FixtureCode_A2Status3 := 2; END_IF;
   #_w4 := "AlwaysTRUE" AND ("AutoProcessData".FixtureCode_A2[4] = "ST10_RecipeDB".ParameterElement.CGlueNGFixtureCode) AND ("AutoProcessData".FixtureCode_A2[4] <> '');
   IF #_w4 THEN "AutoProcessData".GlobalData.FixtureCode_A2Status4 := 1; END_IF;
   IF NOT #_w4 THEN "AutoProcessData".GlobalData.FixtureCode_A2Status4 := 2; END_IF;
   #_w5 := "AlwaysTRUE" AND ("AutoProcessData".FixtureCode_A2[5] = "ST10_RecipeDB".ParameterElement.B2PressCylFixtureCode) AND ("AutoProcessData".FixtureCode_A2[5] <> '');
   IF #_w5 THEN "AutoProcessData".GlobalData.FixtureCode_A2Status5 := 1; END_IF;
   IF NOT #_w5 THEN "AutoProcessData".GlobalData.FixtureCode_A2Status5 := 2; END_IF;
   "AutoProcessData".GlobalData.Fixture2CodeOKFlag := "AlwaysTRUE" AND ((("AutoProcessData".GlobalData.FixtureCode_A2Status1 = 1) AND ("AutoProcessData".GlobalData.FixtureCode_A2Status2 = 1) AND ("AutoProcessData".GlobalData.FixtureCode_A2Status3 = 1) AND ("AutoProcessData".GlobalData.FixtureCode_A2Status4 = 1) AND ("AutoProcessData".GlobalData.FixtureCode_A2Status5 = 1)) OR "ST10_GeneralData".FunctionDeSelect.Global.DeSelectPB_ScanFixture);
END_REGION

REGION Network 23: ChangeOverFinish
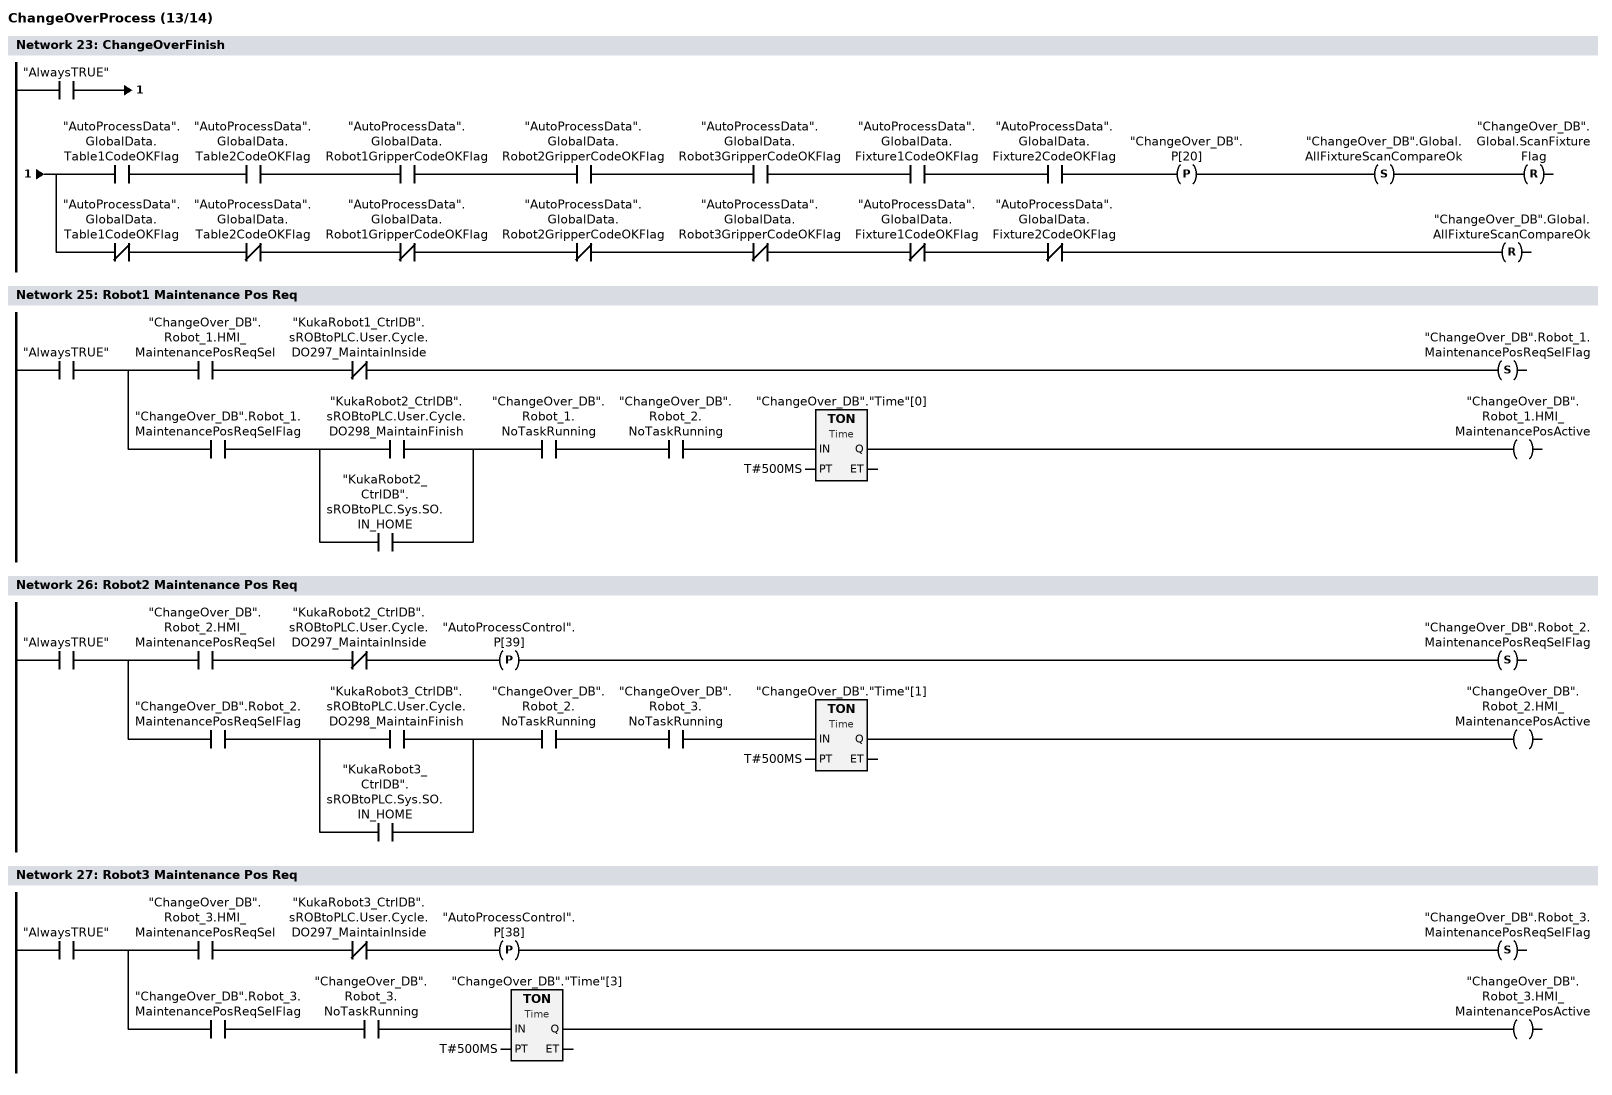
   RUNG wire#powerrail
      Contact( "AlwaysTRUE" )
      wire#w1
      Contact( "AutoProcessData".GlobalData.Table1CodeOKFlag )
      Contact( "AutoProcessData".GlobalData.Table2CodeOKFlag )
      Contact( "AutoProcessData".GlobalData.Robot1GripperCodeOKFlag )
      Contact( "AutoProcessData".GlobalData.Robot2GripperCodeOKFlag )
      Contact( "AutoProcessData".GlobalData.Robot3GripperCodeOKFlag )
      Contact( "AutoProcessData".GlobalData.Fixture1CodeOKFlag )
      Contact( "AutoProcessData".GlobalData.Fixture2CodeOKFlag )
      P_Trig( "ChangeOver_DB".P[20] )
      S_Coil( "ChangeOver_DB".Global.AllFixtureScanCompareOk )
      R_Coil( "ChangeOver_DB".Global.ScanFixtureFlag )
   END_RUNG
   RUNG wire#w1
      I_Contact( "AutoProcessData".GlobalData.Table1CodeOKFlag )
      I_Contact( "AutoProcessData".GlobalData.Table2CodeOKFlag )
      I_Contact( "AutoProcessData".GlobalData.Robot1GripperCodeOKFlag )
      I_Contact( "AutoProcessData".GlobalData.Robot2GripperCodeOKFlag )
      I_Contact( "AutoProcessData".GlobalData.Robot3GripperCodeOKFlag )
      I_Contact( "AutoProcessData".GlobalData.Fixture1CodeOKFlag )
      I_Contact( "AutoProcessData".GlobalData.Fixture2CodeOKFlag )
      R_Coil( "ChangeOver_DB".Global.AllFixtureScanCompareOk )
   END_RUNG
   // the same network as SCL:
   #_w1 := "AlwaysTRUE" AND "AutoProcessData".GlobalData.Table1CodeOKFlag AND "AutoProcessData".GlobalData.Table2CodeOKFlag AND "AutoProcessData".GlobalData.Robot1GripperCodeOKFlag AND "AutoProcessData".GlobalData.Robot2GripperCodeOKFlag AND "AutoProcessData".GlobalData.Robot3GripperCodeOKFlag AND "AutoProcessData".GlobalData.Fixture1CodeOKFlag AND "AutoProcessData".GlobalData.Fixture2CodeOKFlag;
   #_w2 := #_w1 AND NOT "ChangeOver_DB".P[20];   // rising edge
   "ChangeOver_DB".P[20] := #_w1;
   IF #_w2 THEN
       "ChangeOver_DB".Global.AllFixtureScanCompareOk := TRUE;
       "ChangeOver_DB".Global.ScanFixtureFlag := FALSE;
   END_IF;
   IF "AlwaysTRUE" AND NOT "AutoProcessData".GlobalData.Table1CodeOKFlag AND NOT "AutoProcessData".GlobalData.Table2CodeOKFlag AND NOT "AutoProcessData".GlobalData.Robot1GripperCodeOKFlag AND NOT "AutoProcessData".GlobalData.Robot2GripperCodeOKFlag AND NOT "AutoProcessData".GlobalData.Robot3GripperCodeOKFlag AND NOT "AutoProcessData".GlobalData.Fixture1CodeOKFlag AND NOT "AutoProcessData".GlobalData.Fixture2CodeOKFlag THEN
       "ChangeOver_DB".Global.AllFixtureScanCompareOk := FALSE;
   END_IF;
END_REGION

REGION Network 24: ---------------------------------- Manual mode Set maintenance pos / Home pos req ------------------------------------------
END_REGION

